    CONST jointtarget CHANGETOOL:=[[90,0,0,0,-40,0],[9E+09,9E+09,9E+09,9E+09,9E+09,9E+09]];
    TASK PERS wobjdata Pastel_2:=[FALSE,TRUE,"",[[750.001,-195.812,542.432],[0.999786,0.010364,-0.0179194,-3.3711E-5]],[[-815.382,-300.105,150],[0,0.999995,0.00323001,0]]];
    VAR robtarget Target_x_2:=[[0,0,0],[1,0,0,0],[0,0,0,0],[9E+09,9E+09,9E+09,9E+09,9E+09,9E+09]];
    CONST robtarget Aproximacion_2:=[[140.364595003,1.820278874,-22.05975894],[0.119542298,0.027125582,0.159127158,0.979618492],[-1,-1,1,0],[9E+09,9E+09,9E+09,9E+09,9E+09,9E+09]];
    CONST robtarget HOME_2:=[[685.456765267,-392.846667709,72.786791828],[0.784186035,-0.51874833,0.327913883,0.091787349],[0,0,0,0],[9E+09,9E+09,9E+09,9E+09,9E+09,9E+09]];
    CONST robtarget orientacioin_posible_2:=[[21.732086873,134.538800348,-251.768323181],[0.119514706,0.027135826,0.159101077,0.979625811],[-2,0,1,0],[9E+09,9E+09,9E+09,9E+09,9E+09,9E+09]];
    CONST robtarget Target_10_2:=[[139.514118203,143.062380794,-24.987379073],[0.119542298,0.027125582,0.159127158,0.979618492],[-1,-1,1,0],[9E+09,9E+09,9E+09,9E+09,9E+09,9E+09]];
    CONST robtarget Target_20_2:=[[138.975,143.37,0],[0.119542298,0.027125582,0.159127158,0.979618492],[-1,-1,1,0],[9E+09,9E+09,9E+09,9E+09,9E+09,9E+09]];
    CONST robtarget Target_30_2:=[[133.906,143.37,0],[0.119542298,0.027125582,0.159127158,0.979618492],[-1,-1,1,0],[9E+09,9E+09,9E+09,9E+09,9E+09,9E+09]];
    CONST robtarget Target_40_2:=[[126.245,130.656,0],[0.119542298,0.027125582,0.159127158,0.979618492],[-1,-1,1,0],[9E+09,9E+09,9E+09,9E+09,9E+09,9E+09]];
    CONST robtarget Target_50_2:=[[126.245,143.37,0],[0.119542298,0.027125582,0.159127158,0.979618492],[-1,-1,1,0],[9E+09,9E+09,9E+09,9E+09,9E+09,9E+09]];
    CONST robtarget Target_60_2:=[[121.518,143.37,0],[0.119542298,0.027125582,0.159127158,0.979618492],[-1,-1,1,0],[9E+09,9E+09,9E+09,9E+09,9E+09,9E+09]];
    CONST robtarget Target_70_2:=[[121.518,124.69,0],[0.119542298,0.027125582,0.159127158,0.979618492],[-1,-1,1,0],[9E+09,9E+09,9E+09,9E+09,9E+09,9E+09]];
    CONST robtarget Target_80_2:=[[126.603,124.69,0],[0.119542298,0.027125582,0.159127158,0.979618492],[-1,-1,1,0],[9E+09,9E+09,9E+09,9E+09,9E+09,9E+09]];
    CONST robtarget Target_90_2:=[[134.248,137.371,0],[0.119542298,0.027125582,0.159127158,0.979618492],[-1,-1,1,0],[9E+09,9E+09,9E+09,9E+09,9E+09,9E+09]];
    CONST robtarget Target_100_2:=[[134.248,124.69,0],[0.119542298,0.027125582,0.159127158,0.979618492],[-1,-1,1,0],[9E+09,9E+09,9E+09,9E+09,9E+09,9E+09]];
    CONST robtarget Target_110_2:=[[138.975,124.69,0],[0.119542298,0.027125582,0.159127158,0.979618492],[-1,-1,1,0],[9E+09,9E+09,9E+09,9E+09,9E+09,9E+09]];
    CONST robtarget Target_120_2:=[[138.975,143.37,0],[0.119542298,0.027125582,0.159127158,0.979618492],[-1,-1,1,0],[9E+09,9E+09,9E+09,9E+09,9E+09,9E+09]];
    CONST robtarget Target_130_2:=[[138.975,143.37,-10],[0.119542298,0.027125582,0.159127158,0.979618492],[-1,-1,1,0],[9E+09,9E+09,9E+09,9E+09,9E+09,9E+09]];
    CONST robtarget Target_140_2:=[[116.236,143.37,-10],[0.119542298,0.027125582,0.159127158,0.979618492],[-1,-1,1,0],[9E+09,9E+09,9E+09,9E+09,9E+09,9E+09]];
    CONST robtarget Target_150_2:=[[116.236,143.37,0],[0.119542298,0.027125582,0.159127158,0.979618492],[-1,-1,1,0],[9E+09,9E+09,9E+09,9E+09,9E+09,9E+09]];
    CONST robtarget Target_160_2:=[[111.069,143.37,0],[0.119542298,0.027125582,0.159127158,0.979618492],[-1,-1,1,0],[9E+09,9E+09,9E+09,9E+09,9E+09,9E+09]];
    CONST robtarget Target_170_2:=[[111.069,124.69,0],[0.119542298,0.027125582,0.159127158,0.979618492],[-1,-1,1,0],[9E+09,9E+09,9E+09,9E+09,9E+09,9E+09]];
    CONST robtarget Target_180_2:=[[116.236,124.69,0],[0.119542298,0.027125582,0.159127158,0.979618492],[-1,-1,1,0],[9E+09,9E+09,9E+09,9E+09,9E+09,9E+09]];
    CONST robtarget Target_190_2:=[[116.236,143.37,0],[0.119542298,0.027125582,0.159127158,0.979618492],[-1,-1,1,0],[9E+09,9E+09,9E+09,9E+09,9E+09,9E+09]];
    CONST robtarget Target_200_2:=[[116.236,143.37,-10],[0.119542298,0.027125582,0.159127158,0.979618492],[-1,-1,1,0],[9E+09,9E+09,9E+09,9E+09,9E+09,9E+09]];
    CONST robtarget Target_210_2:=[[88.445,137.143,-10],[0.119542298,0.027125582,0.159127158,0.979618492],[-1,-1,1,0],[9E+09,9E+09,9E+09,9E+09,9E+09,9E+09]];
    CONST robtarget Target_220_2:=[[88.445,137.143,0],[0.119542298,0.027125582,0.159127158,0.979618492],[-1,-1,1,0],[9E+09,9E+09,9E+09,9E+09,9E+09,9E+09]];
    CONST robtarget Target_230_2:=[[90.98,142.156,0],[0.119542298,0.027125582,0.159127158,0.979618492],[-1,-1,1,0],[9E+09,9E+09,9E+09,9E+09,9E+09,9E+09]];
    CONST robtarget Target_240_2:=[[96.97,143.973,0],[0.119542298,0.027125582,0.159127158,0.979618492],[-1,-1,1,0],[9E+09,9E+09,9E+09,9E+09,9E+09,9E+09]];
    CONST robtarget Target_250_2:=[[104.06,141.341,0],[0.119542298,0.027125582,0.159127158,0.979618492],[-1,-1,1,0],[9E+09,9E+09,9E+09,9E+09,9E+09,9E+09]];
    CONST robtarget Target_260_2:=[[106.62,134.046,0],[0.119542298,0.027125582,0.159127158,0.979618492],[-1,-1,1,0],[9E+09,9E+09,9E+09,9E+09,9E+09,9E+09]];
    CONST robtarget Target_270_2:=[[104.077,126.752,0],[0.119542298,0.027125582,0.159127158,0.979618492],[-1,-1,1,0],[9E+09,9E+09,9E+09,9E+09,9E+09,9E+09]];
    CONST robtarget Target_280_2:=[[96.954,124.136,0],[0.119542298,0.027125582,0.159127158,0.979618492],[-1,-1,1,0],[9E+09,9E+09,9E+09,9E+09,9E+09,9E+09]];
    CONST robtarget Target_290_2:=[[90.866,125.978,0],[0.119542298,0.027125582,0.159127158,0.979618492],[-1,-1,1,0],[9E+09,9E+09,9E+09,9E+09,9E+09,9E+09]];
    CONST robtarget Target_300_2:=[[88.201,131.178,0],[0.119542298,0.027125582,0.159127158,0.979618492],[-1,-1,1,0],[9E+09,9E+09,9E+09,9E+09,9E+09,9E+09]];
    CONST robtarget Target_310_2:=[[90.556,131.178,0],[0.119542298,0.027125582,0.159127158,0.979618492],[-1,-1,1,0],[9E+09,9E+09,9E+09,9E+09,9E+09,9E+09]];
    CONST robtarget Target_320_2:=[[92.911,131.178,0],[0.119542298,0.027125582,0.159127158,0.979618492],[-1,-1,1,0],[9E+09,9E+09,9E+09,9E+09,9E+09,9E+09]];
    CONST robtarget Target_330_2:=[[94.207,128.781,0],[0.119542298,0.027125582,0.159127158,0.979618492],[-1,-1,1,0],[9E+09,9E+09,9E+09,9E+09,9E+09,9E+09]];
    CONST robtarget Target_340_2:=[[96.937,127.885,0],[0.119542298,0.027125582,0.159127158,0.979618492],[-1,-1,1,0],[9E+09,9E+09,9E+09,9E+09,9E+09,9E+09]];
    CONST robtarget Target_350_2:=[[100.385,129.458,0],[0.119542298,0.027125582,0.159127158,0.979618492],[-1,-1,1,0],[9E+09,9E+09,9E+09,9E+09,9E+09,9E+09]];
    CONST robtarget Target_360_2:=[[101.583,134.03,0],[0.119542298,0.027125582,0.159127158,0.979618492],[-1,-1,1,0],[9E+09,9E+09,9E+09,9E+09,9E+09,9E+09]];
    CONST robtarget Target_370_2:=[[100.426,138.635,0],[0.119542298,0.027125582,0.159127158,0.979618492],[-1,-1,1,0],[9E+09,9E+09,9E+09,9E+09,9E+09,9E+09]];
    CONST robtarget Target_380_2:=[[96.937,140.175,0],[0.119542298,0.027125582,0.159127158,0.979618492],[-1,-1,1,0],[9E+09,9E+09,9E+09,9E+09,9E+09,9E+09]];
    CONST robtarget Target_390_2:=[[94.329,139.376,0],[0.119542298,0.027125582,0.159127158,0.979618492],[-1,-1,1,0],[9E+09,9E+09,9E+09,9E+09,9E+09,9E+09]];
    CONST robtarget Target_400_2:=[[93.058,137.143,0],[0.119542298,0.027125582,0.159127158,0.979618492],[-1,-1,1,0],[9E+09,9E+09,9E+09,9E+09,9E+09,9E+09]];
    CONST robtarget Target_410_2:=[[90.752,137.143,0],[0.119542298,0.027125582,0.159127158,0.979618492],[-1,-1,1,0],[9E+09,9E+09,9E+09,9E+09,9E+09,9E+09]];
    CONST robtarget Target_420_2:=[[88.445,137.143,0],[0.119542298,0.027125582,0.159127158,0.979618492],[-1,-1,1,0],[9E+09,9E+09,9E+09,9E+09,9E+09,9E+09]];
    CONST robtarget Target_430_2:=[[88.445,137.143,-10],[0.119542298,0.027125582,0.159127158,0.979618492],[-1,-1,1,0],[9E+09,9E+09,9E+09,9E+09,9E+09,9E+09]];
    CONST robtarget Target_440_2:=[[65.511,134.046,-10],[0.119542298,0.027125582,0.159127158,0.979618492],[-1,-1,1,0],[9E+09,9E+09,9E+09,9E+09,9E+09,9E+09]];
    CONST robtarget Target_450_2:=[[65.511,134.046,0],[0.119542298,0.027125582,0.159127158,0.979618492],[-1,-1,1,0],[9E+09,9E+09,9E+09,9E+09,9E+09,9E+09]];
    CONST robtarget Target_460_2:=[[68.127,141.3,0],[0.119542298,0.027125582,0.159127158,0.979618492],[-1,-1,1,0],[9E+09,9E+09,9E+09,9E+09,9E+09,9E+09]];
    CONST robtarget Target_470_2:=[[75.21,143.973,0],[0.119542298,0.027125582,0.159127158,0.979618492],[-1,-1,1,0],[9E+09,9E+09,9E+09,9E+09,9E+09,9E+09]];
    CONST robtarget Target_480_2:=[[82.3,141.3,0],[0.119542298,0.027125582,0.159127158,0.979618492],[-1,-1,1,0],[9E+09,9E+09,9E+09,9E+09,9E+09,9E+09]];
    CONST robtarget Target_490_2:=[[84.908,134.046,0],[0.119542298,0.027125582,0.159127158,0.979618492],[-1,-1,1,0],[9E+09,9E+09,9E+09,9E+09,9E+09,9E+09]];
    CONST robtarget Target_500_2:=[[82.3,126.809,0],[0.119542298,0.027125582,0.159127158,0.979618492],[-1,-1,1,0],[9E+09,9E+09,9E+09,9E+09,9E+09,9E+09]];
    CONST robtarget Target_510_2:=[[75.21,124.136,0],[0.119542298,0.027125582,0.159127158,0.979618492],[-1,-1,1,0],[9E+09,9E+09,9E+09,9E+09,9E+09,9E+09]];
    CONST robtarget Target_520_2:=[[68.119,126.809,0],[0.119542298,0.027125582,0.159127158,0.979618492],[-1,-1,1,0],[9E+09,9E+09,9E+09,9E+09,9E+09,9E+09]];
    CONST robtarget Target_530_2:=[[65.511,134.046,0],[0.119542298,0.027125582,0.159127158,0.979618492],[-1,-1,1,0],[9E+09,9E+09,9E+09,9E+09,9E+09,9E+09]];
    CONST robtarget Target_540_2:=[[65.511,134.046,-10],[0.119542298,0.027125582,0.159127158,0.979618492],[-1,-1,1,0],[9E+09,9E+09,9E+09,9E+09,9E+09,9E+09]];
    CONST robtarget Target_550_2:=[[71.298,134.046,-10],[0.119542298,0.027125582,0.159127158,0.979618492],[-1,-1,1,0],[9E+09,9E+09,9E+09,9E+09,9E+09,9E+09]];
    CONST robtarget Target_560_2:=[[71.298,134.046,0],[0.119542298,0.027125582,0.159127158,0.979618492],[-1,-1,1,0],[9E+09,9E+09,9E+09,9E+09,9E+09,9E+09]];
    CONST robtarget Target_570_2:=[[72.235,129.865,0],[0.119542298,0.027125582,0.159127158,0.979618492],[-1,-1,1,0],[9E+09,9E+09,9E+09,9E+09,9E+09,9E+09]];
    CONST robtarget Target_580_2:=[[75.193,128.537,0],[0.119542298,0.027125582,0.159127158,0.979618492],[-1,-1,1,0],[9E+09,9E+09,9E+09,9E+09,9E+09,9E+09]];
    CONST robtarget Target_590_2:=[[78.176,129.865,0],[0.119542298,0.027125582,0.159127158,0.979618492],[-1,-1,1,0],[9E+09,9E+09,9E+09,9E+09,9E+09,9E+09]];
    CONST robtarget Target_600_2:=[[79.122,134.046,0],[0.119542298,0.027125582,0.159127158,0.979618492],[-1,-1,1,0],[9E+09,9E+09,9E+09,9E+09,9E+09,9E+09]];
    CONST robtarget Target_610_2:=[[78.176,138.227,0],[0.119542298,0.027125582,0.159127158,0.979618492],[-1,-1,1,0],[9E+09,9E+09,9E+09,9E+09,9E+09,9E+09]];
    CONST robtarget Target_620_2:=[[75.193,139.556,0],[0.119542298,0.027125582,0.159127158,0.979618492],[-1,-1,1,0],[9E+09,9E+09,9E+09,9E+09,9E+09,9E+09]];
    CONST robtarget Target_630_2:=[[72.235,138.227,0],[0.119542298,0.027125582,0.159127158,0.979618492],[-1,-1,1,0],[9E+09,9E+09,9E+09,9E+09,9E+09,9E+09]];
    CONST robtarget Target_640_2:=[[71.298,134.046,0],[0.119542298,0.027125582,0.159127158,0.979618492],[-1,-1,1,0],[9E+09,9E+09,9E+09,9E+09,9E+09,9E+09]];
    CONST robtarget Target_650_2:=[[71.298,134.046,-10],[0.119542298,0.027125582,0.159127158,0.979618492],[-1,-1,1,0],[9E+09,9E+09,9E+09,9E+09,9E+09,9E+09]];
    CONST robtarget Target_660_2:=[[61.192,143.37,-10],[0.119542298,0.027125582,0.159127158,0.979618492],[-1,-1,1,0],[9E+09,9E+09,9E+09,9E+09,9E+09,9E+09]];
    CONST robtarget Target_670_2:=[[61.192,143.37,0],[0.119542298,0.027125582,0.159127158,0.979618492],[-1,-1,1,0],[9E+09,9E+09,9E+09,9E+09,9E+09,9E+09]];
    CONST robtarget Target_680_2:=[[56.139,143.37,0],[0.119542298,0.027125582,0.159127158,0.979618492],[-1,-1,1,0],[9E+09,9E+09,9E+09,9E+09,9E+09,9E+09]];
    CONST robtarget Target_690_2:=[[56.139,128.7,0],[0.119542298,0.027125582,0.159127158,0.979618492],[-1,-1,1,0],[9E+09,9E+09,9E+09,9E+09,9E+09,9E+09]];
    CONST robtarget Target_700_2:=[[47.402,128.7,0],[0.119542298,0.027125582,0.159127158,0.979618492],[-1,-1,1,0],[9E+09,9E+09,9E+09,9E+09,9E+09,9E+09]];
    CONST robtarget Target_710_2:=[[47.402,124.69,0],[0.119542298,0.027125582,0.159127158,0.979618492],[-1,-1,1,0],[9E+09,9E+09,9E+09,9E+09,9E+09,9E+09]];
    CONST robtarget Target_720_2:=[[61.192,124.69,0],[0.119542298,0.027125582,0.159127158,0.979618492],[-1,-1,1,0],[9E+09,9E+09,9E+09,9E+09,9E+09,9E+09]];
    CONST robtarget Target_730_2:=[[61.192,143.37,0],[0.119542298,0.027125582,0.159127158,0.979618492],[-1,-1,1,0],[9E+09,9E+09,9E+09,9E+09,9E+09,9E+09]];
    CONST robtarget Target_740_2:=[[61.192,143.37,-10],[0.119542298,0.027125582,0.159127158,0.979618492],[-1,-1,1,0],[9E+09,9E+09,9E+09,9E+09,9E+09,9E+09]];
    CONST robtarget Target_750_2:=[[38.567,143.37,-10],[0.119542298,0.027125582,0.159127158,0.979618492],[-1,-1,1,0],[9E+09,9E+09,9E+09,9E+09,9E+09,9E+09]];
    CONST robtarget Target_760_2:=[[38.567,143.37,0],[0.119542298,0.027125582,0.159127158,0.979618492],[-1,-1,1,0],[9E+09,9E+09,9E+09,9E+09,9E+09,9E+09]];
    CONST robtarget Target_770_2:=[[33.025,143.37,0],[0.119542298,0.027125582,0.159127158,0.979618492],[-1,-1,1,0],[9E+09,9E+09,9E+09,9E+09,9E+09,9E+09]];
    CONST robtarget Target_780_2:=[[26.424,124.69,0],[0.119542298,0.027125582,0.159127158,0.979618492],[-1,-1,1,0],[9E+09,9E+09,9E+09,9E+09,9E+09,9E+09]];
    CONST robtarget Target_790_2:=[[31.412,124.69,0],[0.119542298,0.027125582,0.159127158,0.979618492],[-1,-1,1,0],[9E+09,9E+09,9E+09,9E+09,9E+09,9E+09]];
    CONST robtarget Target_800_2:=[[32.178,127.331,0],[0.119542298,0.027125582,0.159127158,0.979618492],[-1,-1,1,0],[9E+09,9E+09,9E+09,9E+09,9E+09,9E+09]];
    CONST robtarget Target_810_2:=[[39.464,127.331,0],[0.119542298,0.027125582,0.159127158,0.979618492],[-1,-1,1,0],[9E+09,9E+09,9E+09,9E+09,9E+09,9E+09]];
    CONST robtarget Target_820_2:=[[40.181,124.69,0],[0.119542298,0.027125582,0.159127158,0.979618492],[-1,-1,1,0],[9E+09,9E+09,9E+09,9E+09,9E+09,9E+09]];
    CONST robtarget Target_830_2:=[[45.169,124.69,0],[0.119542298,0.027125582,0.159127158,0.979618492],[-1,-1,1,0],[9E+09,9E+09,9E+09,9E+09,9E+09,9E+09]];
    CONST robtarget Target_840_2:=[[38.567,143.37,0],[0.119542298,0.027125582,0.159127158,0.979618492],[-1,-1,1,0],[9E+09,9E+09,9E+09,9E+09,9E+09,9E+09]];
    CONST robtarget Target_850_2:=[[38.567,143.37,-10],[0.119542298,0.027125582,0.159127158,0.979618492],[-1,-1,1,0],[9E+09,9E+09,9E+09,9E+09,9E+09,9E+09]];
    CONST robtarget Target_860_2:=[[35.796,138.464,-10],[0.119542298,0.027125582,0.159127158,0.979618492],[-1,-1,1,0],[9E+09,9E+09,9E+09,9E+09,9E+09,9E+09]];
    CONST robtarget Target_870_2:=[[35.796,138.464,0],[0.119542298,0.027125582,0.159127158,0.979618492],[-1,-1,1,0],[9E+09,9E+09,9E+09,9E+09,9E+09,9E+09]];
    CONST robtarget Target_880_2:=[[37.834,130.884,0],[0.119542298,0.027125582,0.159127158,0.979618492],[-1,-1,1,0],[9E+09,9E+09,9E+09,9E+09,9E+09,9E+09]];
    CONST robtarget Target_890_2:=[[33.791,130.884,0],[0.119542298,0.027125582,0.159127158,0.979618492],[-1,-1,1,0],[9E+09,9E+09,9E+09,9E+09,9E+09,9E+09]];
    CONST robtarget Target_900_2:=[[35.796,138.464,0],[0.119542298,0.027125582,0.159127158,0.979618492],[-1,-1,1,0],[9E+09,9E+09,9E+09,9E+09,9E+09,9E+09]];
    CONST robtarget Target_910_2:=[[35.796,138.464,-10],[0.119542298,0.027125582,0.159127158,0.979618492],[-1,-1,1,0],[9E+09,9E+09,9E+09,9E+09,9E+09,9E+09]];
    CONST robtarget Target_920_2:=[[8.038,138.936,-10],[0.119542298,0.027125582,0.159127158,0.979618492],[-1,-1,1,0],[9E+09,9E+09,9E+09,9E+09,9E+09,9E+09]];
    CONST robtarget Target_930_2:=[[8.038,138.936,0],[0.119542298,0.027125582,0.159127158,0.979618492],[-1,-1,1,0],[9E+09,9E+09,9E+09,9E+09,9E+09,9E+09]];
    CONST robtarget Target_940_2:=[[10.58,142.702,0],[0.119542298,0.027125582,0.159127158,0.979618492],[-1,-1,1,0],[9E+09,9E+09,9E+09,9E+09,9E+09,9E+09]];
    CONST robtarget Target_950_2:=[[16.057,143.973,0],[0.119542298,0.027125582,0.159127158,0.979618492],[-1,-1,1,0],[9E+09,9E+09,9E+09,9E+09,9E+09,9E+09]];
    CONST robtarget Target_960_2:=[[21.558,142.416,0],[0.119542298,0.027125582,0.159127158,0.979618492],[-1,-1,1,0],[9E+09,9E+09,9E+09,9E+09,9E+09,9E+09]];
    CONST robtarget Target_970_2:=[[23.588,138.219,0],[0.119542298,0.027125582,0.159127158,0.979618492],[-1,-1,1,0],[9E+09,9E+09,9E+09,9E+09,9E+09,9E+09]];
    CONST robtarget Target_980_2:=[[22.267,134.812,0],[0.119542298,0.027125582,0.159127158,0.979618492],[-1,-1,1,0],[9E+09,9E+09,9E+09,9E+09,9E+09,9E+09]];
    CONST robtarget Target_990_2:=[[16.611,132.4,0],[0.119542298,0.027125582,0.159127158,0.979618492],[-1,-1,1,0],[9E+09,9E+09,9E+09,9E+09,9E+09,9E+09]];
    CONST robtarget Target_1000_2:=[[13.16,131.12,0],[0.119542298,0.027125582,0.159127158,0.979618492],[-1,-1,1,0],[9E+09,9E+09,9E+09,9E+09,9E+09,9E+09]];
    CONST robtarget Target_1010_2:=[[12.324,129.743,0],[0.119542298,0.027125582,0.159127158,0.979618492],[-1,-1,1,0],[9E+09,9E+09,9E+09,9E+09,9E+09,9E+09]];
    CONST robtarget Target_1020_2:=[[13.172,128.17,0],[0.119542298,0.027125582,0.159127158,0.979618492],[-1,-1,1,0],[9E+09,9E+09,9E+09,9E+09,9E+09,9E+09]];
    CONST robtarget Target_1030_2:=[[15.633,127.624,0],[0.119542298,0.027125582,0.159127158,0.979618492],[-1,-1,1,0],[9E+09,9E+09,9E+09,9E+09,9E+09,9E+09]];
    CONST robtarget Target_1040_2:=[[17.858,128.129,0],[0.119542298,0.027125582,0.159127158,0.979618492],[-1,-1,1,0],[9E+09,9E+09,9E+09,9E+09,9E+09,9E+09]];
    CONST robtarget Target_1050_2:=[[18.926,129.629,0],[0.119542298,0.027125582,0.159127158,0.979618492],[-1,-1,1,0],[9E+09,9E+09,9E+09,9E+09,9E+09,9E+09]];
    CONST robtarget Target_1060_2:=[[23.783,129.629,0],[0.119542298,0.027125582,0.159127158,0.979618492],[-1,-1,1,0],[9E+09,9E+09,9E+09,9E+09,9E+09,9E+09]];
    CONST robtarget Target_1070_2:=[[21.192,125.587,0],[0.119542298,0.027125582,0.159127158,0.979618492],[-1,-1,1,0],[9E+09,9E+09,9E+09,9E+09,9E+09,9E+09]];
    CONST robtarget Target_1080_2:=[[15.715,124.169,0],[0.119542298,0.027125582,0.159127158,0.979618492],[-1,-1,1,0],[9E+09,9E+09,9E+09,9E+09,9E+09,9E+09]];
    CONST robtarget Target_1090_2:=[[9.554,125.741,0],[0.119542298,0.027125582,0.159127158,0.979618492],[-1,-1,1,0],[9E+09,9E+09,9E+09,9E+09,9E+09,9E+09]];
    CONST robtarget Target_1100_2:=[[7.451,130.379,0],[0.119542298,0.027125582,0.159127158,0.979618492],[-1,-1,1,0],[9E+09,9E+09,9E+09,9E+09,9E+09,9E+09]];
    CONST robtarget Target_1110_2:=[[8.885,133.875,0],[0.119542298,0.027125582,0.159127158,0.979618492],[-1,-1,1,0],[9E+09,9E+09,9E+09,9E+09,9E+09,9E+09]];
    CONST robtarget Target_1120_2:=[[15.03,136.328,0],[0.119542298,0.027125582,0.159127158,0.979618492],[-1,-1,1,0],[9E+09,9E+09,9E+09,9E+09,9E+09,9E+09]];
    CONST robtarget Target_1130_2:=[[17.85,137.412,0],[0.119542298,0.027125582,0.159127158,0.979618492],[-1,-1,1,0],[9E+09,9E+09,9E+09,9E+09,9E+09,9E+09]];
    CONST robtarget Target_1140_2:=[[18.698,138.773,0],[0.119542298,0.027125582,0.159127158,0.979618492],[-1,-1,1,0],[9E+09,9E+09,9E+09,9E+09,9E+09,9E+09]];
    CONST robtarget Target_1150_2:=[[17.972,140.208,0],[0.119542298,0.027125582,0.159127158,0.979618492],[-1,-1,1,0],[9E+09,9E+09,9E+09,9E+09,9E+09,9E+09]];
    CONST robtarget Target_1160_2:=[[15.976,140.729,0],[0.119542298,0.027125582,0.159127158,0.979618492],[-1,-1,1,0],[9E+09,9E+09,9E+09,9E+09,9E+09,9E+09]];
    CONST robtarget Target_1170_2:=[[13.889,140.265,0],[0.119542298,0.027125582,0.159127158,0.979618492],[-1,-1,1,0],[9E+09,9E+09,9E+09,9E+09,9E+09,9E+09]];
    CONST robtarget Target_1180_2:=[[12.879,138.936,0],[0.119542298,0.027125582,0.159127158,0.979618492],[-1,-1,1,0],[9E+09,9E+09,9E+09,9E+09,9E+09,9E+09]];
    CONST robtarget Target_1190_2:=[[8.038,138.936,0],[0.119542298,0.027125582,0.159127158,0.979618492],[-1,-1,1,0],[9E+09,9E+09,9E+09,9E+09,9E+09,9E+09]];
    CONST robtarget Target_1200_2:=[[8.038,138.936,-10],[0.119542298,0.027125582,0.159127158,0.979618492],[-1,-1,1,0],[9E+09,9E+09,9E+09,9E+09,9E+09,9E+09]];
    CONST robtarget Target_1210_2:=[[113.571,103.208,-10],[0.119542298,0.027125582,0.159127158,0.979618492],[-1,-1,1,0],[9E+09,9E+09,9E+09,9E+09,9E+09,9E+09]];
    CONST robtarget Target_1220_2:=[[113.571,103.208,0],[0.119542298,0.027125582,0.159127158,0.979618492],[-1,-1,1,0],[9E+09,9E+09,9E+09,9E+09,9E+09,9E+09]];
    CONST robtarget Target_1230_2:=[[116.106,108.22,0],[0.119542298,0.027125582,0.159127158,0.979618492],[-1,-1,1,0],[9E+09,9E+09,9E+09,9E+09,9E+09,9E+09]];
    CONST robtarget Target_1240_2:=[[122.096,110.037,0],[0.119542298,0.027125582,0.159127158,0.979618492],[-1,-1,1,0],[9E+09,9E+09,9E+09,9E+09,9E+09,9E+09]];
    CONST robtarget Target_1250_2:=[[129.187,107.405,0],[0.119542298,0.027125582,0.159127158,0.979618492],[-1,-1,1,0],[9E+09,9E+09,9E+09,9E+09,9E+09,9E+09]];
    CONST robtarget Target_1260_2:=[[131.746,100.111,0],[0.119542298,0.027125582,0.159127158,0.979618492],[-1,-1,1,0],[9E+09,9E+09,9E+09,9E+09,9E+09,9E+09]];
    CONST robtarget Target_1270_2:=[[129.203,92.817,0],[0.119542298,0.027125582,0.159127158,0.979618492],[-1,-1,1,0],[9E+09,9E+09,9E+09,9E+09,9E+09,9E+09]];
    CONST robtarget Target_1280_2:=[[122.08,90.2,0],[0.119542298,0.027125582,0.159127158,0.979618492],[-1,-1,1,0],[9E+09,9E+09,9E+09,9E+09,9E+09,9E+09]];
    CONST robtarget Target_1290_2:=[[115.992,92.042,0],[0.119542298,0.027125582,0.159127158,0.979618492],[-1,-1,1,0],[9E+09,9E+09,9E+09,9E+09,9E+09,9E+09]];
    CONST robtarget Target_1300_2:=[[113.327,97.242,0],[0.119542298,0.027125582,0.159127158,0.979618492],[-1,-1,1,0],[9E+09,9E+09,9E+09,9E+09,9E+09,9E+09]];
    CONST robtarget Target_1310_2:=[[118.038,97.242,0],[0.119542298,0.027125582,0.159127158,0.979618492],[-1,-1,1,0],[9E+09,9E+09,9E+09,9E+09,9E+09,9E+09]];
    CONST robtarget Target_1320_2:=[[119.333,94.846,0],[0.119542298,0.027125582,0.159127158,0.979618492],[-1,-1,1,0],[9E+09,9E+09,9E+09,9E+09,9E+09,9E+09]];
    CONST robtarget Target_1330_2:=[[122.064,93.949,0],[0.119542298,0.027125582,0.159127158,0.979618492],[-1,-1,1,0],[9E+09,9E+09,9E+09,9E+09,9E+09,9E+09]];
    CONST robtarget Target_1340_2:=[[125.511,95.522,0],[0.119542298,0.027125582,0.159127158,0.979618492],[-1,-1,1,0],[9E+09,9E+09,9E+09,9E+09,9E+09,9E+09]];
    CONST robtarget Target_1350_2:=[[126.709,100.094,0],[0.119542298,0.027125582,0.159127158,0.979618492],[-1,-1,1,0],[9E+09,9E+09,9E+09,9E+09,9E+09,9E+09]];
    CONST robtarget Target_1360_2:=[[125.552,104.699,0],[0.119542298,0.027125582,0.159127158,0.979618492],[-1,-1,1,0],[9E+09,9E+09,9E+09,9E+09,9E+09,9E+09]];
    CONST robtarget Target_1370_2:=[[122.064,106.239,0],[0.119542298,0.027125582,0.159127158,0.979618492],[-1,-1,1,0],[9E+09,9E+09,9E+09,9E+09,9E+09,9E+09]];
    CONST robtarget Target_1380_2:=[[119.456,105.441,0],[0.119542298,0.027125582,0.159127158,0.979618492],[-1,-1,1,0],[9E+09,9E+09,9E+09,9E+09,9E+09,9E+09]];
    CONST robtarget Target_1390_2:=[[118.184,103.208,0],[0.119542298,0.027125582,0.159127158,0.979618492],[-1,-1,1,0],[9E+09,9E+09,9E+09,9E+09,9E+09,9E+09]];
    CONST robtarget Target_1400_2:=[[113.571,103.208,0],[0.119542298,0.027125582,0.159127158,0.979618492],[-1,-1,1,0],[9E+09,9E+09,9E+09,9E+09,9E+09,9E+09]];
    CONST robtarget Target_1410_2:=[[113.571,103.208,-10],[0.119542298,0.027125582,0.159127158,0.979618492],[-1,-1,1,0],[9E+09,9E+09,9E+09,9E+09,9E+09,9E+09]];
    CONST robtarget Target_1420_2:=[[98.771,109.434,-10],[0.119542298,0.027125582,0.159127158,0.979618492],[-1,-1,1,0],[9E+09,9E+09,9E+09,9E+09,9E+09,9E+09]];
    CONST robtarget Target_1430_2:=[[98.771,109.434,0],[0.119542298,0.027125582,0.159127158,0.979618492],[-1,-1,1,0],[9E+09,9E+09,9E+09,9E+09,9E+09,9E+09]];
    CONST robtarget Target_1440_2:=[[92.17,90.755,0],[0.119542298,0.027125582,0.159127158,0.979618492],[-1,-1,1,0],[9E+09,9E+09,9E+09,9E+09,9E+09,9E+09]];
    CONST robtarget Target_1450_2:=[[97.157,90.755,0],[0.119542298,0.027125582,0.159127158,0.979618492],[-1,-1,1,0],[9E+09,9E+09,9E+09,9E+09,9E+09,9E+09]];
    CONST robtarget Target_1460_2:=[[97.924,93.395,0],[0.119542298,0.027125582,0.159127158,0.979618492],[-1,-1,1,0],[9E+09,9E+09,9E+09,9E+09,9E+09,9E+09]];
    CONST robtarget Target_1470_2:=[[105.21,93.395,0],[0.119542298,0.027125582,0.159127158,0.979618492],[-1,-1,1,0],[9E+09,9E+09,9E+09,9E+09,9E+09,9E+09]];
    CONST robtarget Target_1480_2:=[[105.927,90.755,0],[0.119542298,0.027125582,0.159127158,0.979618492],[-1,-1,1,0],[9E+09,9E+09,9E+09,9E+09,9E+09,9E+09]];
    CONST robtarget Target_1490_2:=[[110.915,90.755,0],[0.119542298,0.027125582,0.159127158,0.979618492],[-1,-1,1,0],[9E+09,9E+09,9E+09,9E+09,9E+09,9E+09]];
    CONST robtarget Target_1500_2:=[[104.313,109.434,0],[0.119542298,0.027125582,0.159127158,0.979618492],[-1,-1,1,0],[9E+09,9E+09,9E+09,9E+09,9E+09,9E+09]];
    CONST robtarget Target_1510_2:=[[98.771,109.434,0],[0.119542298,0.027125582,0.159127158,0.979618492],[-1,-1,1,0],[9E+09,9E+09,9E+09,9E+09,9E+09,9E+09]];
    CONST robtarget Target_1520_2:=[[98.771,109.434,-10],[0.119542298,0.027125582,0.159127158,0.979618492],[-1,-1,1,0],[9E+09,9E+09,9E+09,9E+09,9E+09,9E+09]];
    CONST robtarget Target_1530_2:=[[101.542,104.528,-10],[0.119542298,0.027125582,0.159127158,0.979618492],[-1,-1,1,0],[9E+09,9E+09,9E+09,9E+09,9E+09,9E+09]];
    CONST robtarget Target_1540_2:=[[101.542,104.528,0],[0.119542298,0.027125582,0.159127158,0.979618492],[-1,-1,1,0],[9E+09,9E+09,9E+09,9E+09,9E+09,9E+09]];
    CONST robtarget Target_1550_2:=[[103.58,96.949,0],[0.119542298,0.027125582,0.159127158,0.979618492],[-1,-1,1,0],[9E+09,9E+09,9E+09,9E+09,9E+09,9E+09]];
    CONST robtarget Target_1560_2:=[[99.537,96.949,0],[0.119542298,0.027125582,0.159127158,0.979618492],[-1,-1,1,0],[9E+09,9E+09,9E+09,9E+09,9E+09,9E+09]];
    CONST robtarget Target_1570_2:=[[101.542,104.528,0],[0.119542298,0.027125582,0.159127158,0.979618492],[-1,-1,1,0],[9E+09,9E+09,9E+09,9E+09,9E+09,9E+09]];
    CONST robtarget Target_1580_2:=[[101.542,104.528,-10],[0.119542298,0.027125582,0.159127158,0.979618492],[-1,-1,1,0],[9E+09,9E+09,9E+09,9E+09,9E+09,9E+09]];
    CONST robtarget Target_1590_2:=[[88.747,109.434,-10],[0.119542298,0.027125582,0.159127158,0.979618492],[-1,-1,1,0],[9E+09,9E+09,9E+09,9E+09,9E+09,9E+09]];
    CONST robtarget Target_1600_2:=[[88.747,109.434,0],[0.119542298,0.027125582,0.159127158,0.979618492],[-1,-1,1,0],[9E+09,9E+09,9E+09,9E+09,9E+09,9E+09]];
    CONST robtarget Target_1610_2:=[[88.747,90.755,0],[0.119542298,0.027125582,0.159127158,0.979618492],[-1,-1,1,0],[9E+09,9E+09,9E+09,9E+09,9E+09,9E+09]];
    CONST robtarget Target_1620_2:=[[84.297,90.755,0],[0.119542298,0.027125582,0.159127158,0.979618492],[-1,-1,1,0],[9E+09,9E+09,9E+09,9E+09,9E+09,9E+09]];
    CONST robtarget Target_1630_2:=[[84.297,105.848,0],[0.119542298,0.027125582,0.159127158,0.979618492],[-1,-1,1,0],[9E+09,9E+09,9E+09,9E+09,9E+09,9E+09]];
    CONST robtarget Target_1640_2:=[[83.743,105.848,0],[0.119542298,0.027125582,0.159127158,0.979618492],[-1,-1,1,0],[9E+09,9E+09,9E+09,9E+09,9E+09,9E+09]];
    CONST robtarget Target_1650_2:=[[79.88,90.755,0],[0.119542298,0.027125582,0.159127158,0.979618492],[-1,-1,1,0],[9E+09,9E+09,9E+09,9E+09,9E+09,9E+09]];
    CONST robtarget Target_1660_2:=[[76.424,90.755,0],[0.119542298,0.027125582,0.159127158,0.979618492],[-1,-1,1,0],[9E+09,9E+09,9E+09,9E+09,9E+09,9E+09]];
    CONST robtarget Target_1670_2:=[[72.626,105.848,0],[0.119542298,0.027125582,0.159127158,0.979618492],[-1,-1,1,0],[9E+09,9E+09,9E+09,9E+09,9E+09,9E+09]];
    CONST robtarget Target_1680_2:=[[71.941,105.848,0],[0.119542298,0.027125582,0.159127158,0.979618492],[-1,-1,1,0],[9E+09,9E+09,9E+09,9E+09,9E+09,9E+09]];
    CONST robtarget Target_1690_2:=[[71.941,90.755,0],[0.119542298,0.027125582,0.159127158,0.979618492],[-1,-1,1,0],[9E+09,9E+09,9E+09,9E+09,9E+09,9E+09]];
    CONST robtarget Target_1700_2:=[[67.557,90.755,0],[0.119542298,0.027125582,0.159127158,0.979618492],[-1,-1,1,0],[9E+09,9E+09,9E+09,9E+09,9E+09,9E+09]];
    CONST robtarget Target_1710_2:=[[67.557,109.434,0],[0.119542298,0.027125582,0.159127158,0.979618492],[-1,-1,1,0],[9E+09,9E+09,9E+09,9E+09,9E+09,9E+09]];
    CONST robtarget Target_1720_2:=[[74.175,109.434,0],[0.119542298,0.027125582,0.159127158,0.979618492],[-1,-1,1,0],[9E+09,9E+09,9E+09,9E+09,9E+09,9E+09]];
    CONST robtarget Target_1730_2:=[[78.152,95.482,0],[0.119542298,0.027125582,0.159127158,0.979618492],[-1,-1,1,0],[9E+09,9E+09,9E+09,9E+09,9E+09,9E+09]];
    CONST robtarget Target_1740_2:=[[82.113,109.434,0],[0.119542298,0.027125582,0.159127158,0.979618492],[-1,-1,1,0],[9E+09,9E+09,9E+09,9E+09,9E+09,9E+09]];
    CONST robtarget Target_1750_2:=[[88.747,109.434,0],[0.119542298,0.027125582,0.159127158,0.979618492],[-1,-1,1,0],[9E+09,9E+09,9E+09,9E+09,9E+09,9E+09]];
    CONST robtarget Target_1760_2:=[[88.747,109.434,-10],[0.119542298,0.027125582,0.159127158,0.979618492],[-1,-1,1,0],[9E+09,9E+09,9E+09,9E+09,9E+09,9E+09]];
    CONST robtarget Target_1770_2:=[[62.308,109.434,-10],[0.119542298,0.027125582,0.159127158,0.979618492],[-1,-1,1,0],[9E+09,9E+09,9E+09,9E+09,9E+09,9E+09]];
    CONST robtarget Target_1780_2:=[[62.308,109.434,0],[0.119542298,0.027125582,0.159127158,0.979618492],[-1,-1,1,0],[9E+09,9E+09,9E+09,9E+09,9E+09,9E+09]];
    CONST robtarget Target_1790_2:=[[62.308,90.755,0],[0.119542298,0.027125582,0.159127158,0.979618492],[-1,-1,1,0],[9E+09,9E+09,9E+09,9E+09,9E+09,9E+09]];
    CONST robtarget Target_1800_2:=[[57.141,90.755,0],[0.119542298,0.027125582,0.159127158,0.979618492],[-1,-1,1,0],[9E+09,9E+09,9E+09,9E+09,9E+09,9E+09]];
    CONST robtarget Target_1810_2:=[[57.141,109.434,0],[0.119542298,0.027125582,0.159127158,0.979618492],[-1,-1,1,0],[9E+09,9E+09,9E+09,9E+09,9E+09,9E+09]];
    CONST robtarget Target_1820_2:=[[62.308,109.434,0],[0.119542298,0.027125582,0.159127158,0.979618492],[-1,-1,1,0],[9E+09,9E+09,9E+09,9E+09,9E+09,9E+09]];
    CONST robtarget Target_1830_2:=[[62.308,109.434,-10],[0.119542298,0.027125582,0.159127158,0.979618492],[-1,-1,1,0],[9E+09,9E+09,9E+09,9E+09,9E+09,9E+09]];
    CONST robtarget Target_1840_2:=[[51.86,109.434,-10],[0.119542298,0.027125582,0.159127158,0.979618492],[-1,-1,1,0],[9E+09,9E+09,9E+09,9E+09,9E+09,9E+09]];
    CONST robtarget Target_1850_2:=[[51.86,109.434,0],[0.119542298,0.027125582,0.159127158,0.979618492],[-1,-1,1,0],[9E+09,9E+09,9E+09,9E+09,9E+09,9E+09]];
    CONST robtarget Target_1860_2:=[[51.86,90.755,0],[0.119542298,0.027125582,0.159127158,0.979618492],[-1,-1,1,0],[9E+09,9E+09,9E+09,9E+09,9E+09,9E+09]];
    CONST robtarget Target_1870_2:=[[38.07,90.755,0],[0.119542298,0.027125582,0.159127158,0.979618492],[-1,-1,1,0],[9E+09,9E+09,9E+09,9E+09,9E+09,9E+09]];
    CONST robtarget Target_1880_2:=[[38.07,94.764,0],[0.119542298,0.027125582,0.159127158,0.979618492],[-1,-1,1,0],[9E+09,9E+09,9E+09,9E+09,9E+09,9E+09]];
    CONST robtarget Target_1890_2:=[[46.807,94.764,0],[0.119542298,0.027125582,0.159127158,0.979618492],[-1,-1,1,0],[9E+09,9E+09,9E+09,9E+09,9E+09,9E+09]];
    CONST robtarget Target_1900_2:=[[46.807,109.434,0],[0.119542298,0.027125582,0.159127158,0.979618492],[-1,-1,1,0],[9E+09,9E+09,9E+09,9E+09,9E+09,9E+09]];
    CONST robtarget Target_1910_2:=[[51.86,109.434,0],[0.119542298,0.027125582,0.159127158,0.979618492],[-1,-1,1,0],[9E+09,9E+09,9E+09,9E+09,9E+09,9E+09]];
    CONST robtarget Target_1920_2:=[[51.86,109.434,-10],[0.119542298,0.027125582,0.159127158,0.979618492],[-1,-1,1,0],[9E+09,9E+09,9E+09,9E+09,9E+09,9E+09]];
    CONST robtarget Target_1930_2:=[[25.242,106.256,-10],[0.119542298,0.027125582,0.159127158,0.979618492],[-1,-1,1,0],[9E+09,9E+09,9E+09,9E+09,9E+09,9E+09]];
    CONST robtarget Target_1940_2:=[[25.242,106.256,0],[0.119542298,0.027125582,0.159127158,0.979618492],[-1,-1,1,0],[9E+09,9E+09,9E+09,9E+09,9E+09,9E+09]];
    CONST robtarget Target_1950_2:=[[28.739,104.772,0],[0.119542298,0.027125582,0.159127158,0.979618492],[-1,-1,1,0],[9E+09,9E+09,9E+09,9E+09,9E+09,9E+09]];
    CONST robtarget Target_1960_2:=[[29.855,100.111,0],[0.119542298,0.027125582,0.159127158,0.979618492],[-1,-1,1,0],[9E+09,9E+09,9E+09,9E+09,9E+09,9E+09]];
    CONST robtarget Target_1970_2:=[[28.739,95.449,0],[0.119542298,0.027125582,0.159127158,0.979618492],[-1,-1,1,0],[9E+09,9E+09,9E+09,9E+09,9E+09,9E+09]];
    CONST robtarget Target_1980_2:=[[25.242,93.966,0],[0.119542298,0.027125582,0.159127158,0.979618492],[-1,-1,1,0],[9E+09,9E+09,9E+09,9E+09,9E+09,9E+09]];
    CONST robtarget Target_1990_2:=[[21.754,95.441,0],[0.119542298,0.027125582,0.159127158,0.979618492],[-1,-1,1,0],[9E+09,9E+09,9E+09,9E+09,9E+09,9E+09]];
    CONST robtarget Target_2000_2:=[[20.646,100.111,0],[0.119542298,0.027125582,0.159127158,0.979618492],[-1,-1,1,0],[9E+09,9E+09,9E+09,9E+09,9E+09,9E+09]];
    CONST robtarget Target_2010_2:=[[21.754,104.772,0],[0.119542298,0.027125582,0.159127158,0.979618492],[-1,-1,1,0],[9E+09,9E+09,9E+09,9E+09,9E+09,9E+09]];
    CONST robtarget Target_2020_2:=[[25.242,106.256,0],[0.119542298,0.027125582,0.159127158,0.979618492],[-1,-1,1,0],[9E+09,9E+09,9E+09,9E+09,9E+09,9E+09]];
    CONST robtarget Target_2030_2:=[[25.242,106.256,-10],[0.119542298,0.027125582,0.159127158,0.979618492],[-1,-1,1,0],[9E+09,9E+09,9E+09,9E+09,9E+09,9E+09]];
    CONST robtarget Target_2040_2:=[[25.258,110.037,-10],[0.119542298,0.027125582,0.159127158,0.979618492],[-1,-1,1,0],[9E+09,9E+09,9E+09,9E+09,9E+09,9E+09]];
    CONST robtarget Target_2050_2:=[[25.258,110.037,0],[0.119542298,0.027125582,0.159127158,0.979618492],[-1,-1,1,0],[9E+09,9E+09,9E+09,9E+09,9E+09,9E+09]];
    CONST robtarget Target_2060_2:=[[18.176,107.364,0],[0.119542298,0.027125582,0.159127158,0.979618492],[-1,-1,1,0],[9E+09,9E+09,9E+09,9E+09,9E+09,9E+09]];
    CONST robtarget Target_2070_2:=[[15.56,100.111,0],[0.119542298,0.027125582,0.159127158,0.979618492],[-1,-1,1,0],[9E+09,9E+09,9E+09,9E+09,9E+09,9E+09]];
    CONST robtarget Target_2080_2:=[[18.168,92.874,0],[0.119542298,0.027125582,0.159127158,0.979618492],[-1,-1,1,0],[9E+09,9E+09,9E+09,9E+09,9E+09,9E+09]];
    CONST robtarget Target_2090_2:=[[25.258,90.2,0],[0.119542298,0.027125582,0.159127158,0.979618492],[-1,-1,1,0],[9E+09,9E+09,9E+09,9E+09,9E+09,9E+09]];
    CONST robtarget Target_2100_2:=[[32.349,92.874,0],[0.119542298,0.027125582,0.159127158,0.979618492],[-1,-1,1,0],[9E+09,9E+09,9E+09,9E+09,9E+09,9E+09]];
    CONST robtarget Target_2110_2:=[[34.957,100.111,0],[0.119542298,0.027125582,0.159127158,0.979618492],[-1,-1,1,0],[9E+09,9E+09,9E+09,9E+09,9E+09,9E+09]];
    CONST robtarget Target_2120_2:=[[32.349,107.364,0],[0.119542298,0.027125582,0.159127158,0.979618492],[-1,-1,1,0],[9E+09,9E+09,9E+09,9E+09,9E+09,9E+09]];
    CONST robtarget Target_2130_2:=[[25.258,110.037,0],[0.119542298,0.027125582,0.159127158,0.979618492],[-1,-1,1,0],[9E+09,9E+09,9E+09,9E+09,9E+09,9E+09]];
    CONST robtarget Target_2140_2:=[[25.258,110.037,-10],[0.119542298,0.027125582,0.159127158,0.979618492],[-1,-1,1,0],[9E+09,9E+09,9E+09,9E+09,9E+09,9E+09]];
    CONST robtarget Target_2150_2:=[[120.369,69.924,-10],[0.119542298,0.027125582,0.159127158,0.979618492],[-1,-1,1,0],[9E+09,9E+09,9E+09,9E+09,9E+09,9E+09]];
    CONST robtarget Target_2160_2:=[[120.369,69.924,0],[0.119542298,0.027125582,0.159127158,0.979618492],[-1,-1,1,0],[9E+09,9E+09,9E+09,9E+09,9E+09,9E+09]];
    CONST robtarget Target_2170_2:=[[125.21,69.924,0],[0.119542298,0.027125582,0.159127158,0.979618492],[-1,-1,1,0],[9E+09,9E+09,9E+09,9E+09,9E+09,9E+09]];
    CONST robtarget Target_2180_2:=[[126.514,71.717,0],[0.119542298,0.027125582,0.159127158,0.979618492],[-1,-1,1,0],[9E+09,9E+09,9E+09,9E+09,9E+09,9E+09]];
    CONST robtarget Target_2190_2:=[[128.763,72.337,0],[0.119542298,0.027125582,0.159127158,0.979618492],[-1,-1,1,0],[9E+09,9E+09,9E+09,9E+09,9E+09,9E+09]];
    CONST robtarget Target_2200_2:=[[132.178,70.715,0],[0.119542298,0.027125582,0.159127158,0.979618492],[-1,-1,1,0],[9E+09,9E+09,9E+09,9E+09,9E+09,9E+09]];
    CONST robtarget Target_2210_2:=[[133.376,66.061,0],[0.119542298,0.027125582,0.159127158,0.979618492],[-1,-1,1,0],[9E+09,9E+09,9E+09,9E+09,9E+09,9E+09]];
    CONST robtarget Target_2220_2:=[[132.243,61.367,0],[0.119542298,0.027125582,0.159127158,0.979618492],[-1,-1,1,0],[9E+09,9E+09,9E+09,9E+09,9E+09,9E+09]];
    CONST robtarget Target_2230_2:=[[128.763,59.834,0],[0.119542298,0.027125582,0.159127158,0.979618492],[-1,-1,1,0],[9E+09,9E+09,9E+09,9E+09,9E+09,9E+09]];
    CONST robtarget Target_2240_2:=[[125.723,60.861,0],[0.119542298,0.027125582,0.159127158,0.979618492],[-1,-1,1,0],[9E+09,9E+09,9E+09,9E+09,9E+09,9E+09]];
    CONST robtarget Target_2250_2:=[[124.46,63.486,0],[0.119542298,0.027125582,0.159127158,0.979618492],[-1,-1,1,0],[9E+09,9E+09,9E+09,9E+09,9E+09,9E+09]];
    CONST robtarget Target_2260_2:=[[125.927,63.494,0],[0.119542298,0.027125582,0.159127158,0.979618492],[-1,-1,1,0],[9E+09,9E+09,9E+09,9E+09,9E+09,9E+09]];
    CONST robtarget Target_2270_2:=[[127.394,63.502,0],[0.119542298,0.027125582,0.159127158,0.979618492],[-1,-1,1,0],[9E+09,9E+09,9E+09,9E+09,9E+09,9E+09]];
    CONST robtarget Target_2280_2:=[[127.394,66.501,0],[0.119542298,0.027125582,0.159127158,0.979618492],[-1,-1,1,0],[9E+09,9E+09,9E+09,9E+09,9E+09,9E+09]];
    CONST robtarget Target_2290_2:=[[119.961,66.501,0],[0.119542298,0.027125582,0.159127158,0.979618492],[-1,-1,1,0],[9E+09,9E+09,9E+09,9E+09,9E+09,9E+09]];
    CONST robtarget Target_2300_2:=[[119.961,56.819,0],[0.119542298,0.027125582,0.159127158,0.979618492],[-1,-1,1,0],[9E+09,9E+09,9E+09,9E+09,9E+09,9E+09]];
    CONST robtarget Target_2310_2:=[[122.928,56.819,0],[0.119542298,0.027125582,0.159127158,0.979618492],[-1,-1,1,0],[9E+09,9E+09,9E+09,9E+09,9E+09,9E+09]];
    CONST robtarget Target_2320_2:=[[123.433,59.557,0],[0.119542298,0.027125582,0.159127158,0.979618492],[-1,-1,1,0],[9E+09,9E+09,9E+09,9E+09,9E+09,9E+09]];
    CONST robtarget Target_2330_2:=[[125.78,57.129,0],[0.119542298,0.027125582,0.159127158,0.979618492],[-1,-1,1,0],[9E+09,9E+09,9E+09,9E+09,9E+09,9E+09]];
    CONST robtarget Target_2340_2:=[[129.855,56.265,0],[0.119542298,0.027125582,0.159127158,0.979618492],[-1,-1,1,0],[9E+09,9E+09,9E+09,9E+09,9E+09,9E+09]];
    CONST robtarget Target_2350_2:=[[136.155,58.938,0],[0.119542298,0.027125582,0.159127158,0.979618492],[-1,-1,1,0],[9E+09,9E+09,9E+09,9E+09,9E+09,9E+09]];
    CONST robtarget Target_2360_2:=[[138.478,66.175,0],[0.119542298,0.027125582,0.159127158,0.979618492],[-1,-1,1,0],[9E+09,9E+09,9E+09,9E+09,9E+09,9E+09]];
    CONST robtarget Target_2370_2:=[[135.91,73.469,0],[0.119542298,0.027125582,0.159127158,0.979618492],[-1,-1,1,0],[9E+09,9E+09,9E+09,9E+09,9E+09,9E+09]];
    CONST robtarget Target_2380_2:=[[128.796,76.102,0],[0.119542298,0.027125582,0.159127158,0.979618492],[-1,-1,1,0],[9E+09,9E+09,9E+09,9E+09,9E+09,9E+09]];
    CONST robtarget Target_2390_2:=[[123.148,74.48,0],[0.119542298,0.027125582,0.159127158,0.979618492],[-1,-1,1,0],[9E+09,9E+09,9E+09,9E+09,9E+09,9E+09]];
    CONST robtarget Target_2400_2:=[[120.369,69.924,0],[0.119542298,0.027125582,0.159127158,0.979618492],[-1,-1,1,0],[9E+09,9E+09,9E+09,9E+09,9E+09,9E+09]];
    CONST robtarget Target_2410_2:=[[120.369,69.924,-10],[0.119542298,0.027125582,0.159127158,0.979618492],[-1,-1,1,0],[9E+09,9E+09,9E+09,9E+09,9E+09,9E+09]];
    CONST robtarget Target_2420_2:=[[110.1,75.499,-10],[0.119542298,0.027125582,0.159127158,0.979618492],[-1,-1,1,0],[9E+09,9E+09,9E+09,9E+09,9E+09,9E+09]];
    CONST robtarget Target_2430_2:=[[110.1,75.499,0],[0.119542298,0.027125582,0.159127158,0.979618492],[-1,-1,1,0],[9E+09,9E+09,9E+09,9E+09,9E+09,9E+09]];
    CONST robtarget Target_2440_2:=[[104.558,75.499,0],[0.119542298,0.027125582,0.159127158,0.979618492],[-1,-1,1,0],[9E+09,9E+09,9E+09,9E+09,9E+09,9E+09]];
    CONST robtarget Target_2450_2:=[[97.956,56.819,0],[0.119542298,0.027125582,0.159127158,0.979618492],[-1,-1,1,0],[9E+09,9E+09,9E+09,9E+09,9E+09,9E+09]];
    CONST robtarget Target_2460_2:=[[102.944,56.819,0],[0.119542298,0.027125582,0.159127158,0.979618492],[-1,-1,1,0],[9E+09,9E+09,9E+09,9E+09,9E+09,9E+09]];
    CONST robtarget Target_2470_2:=[[103.71,59.46,0],[0.119542298,0.027125582,0.159127158,0.979618492],[-1,-1,1,0],[9E+09,9E+09,9E+09,9E+09,9E+09,9E+09]];
    CONST robtarget Target_2480_2:=[[110.996,59.46,0],[0.119542298,0.027125582,0.159127158,0.979618492],[-1,-1,1,0],[9E+09,9E+09,9E+09,9E+09,9E+09,9E+09]];
    CONST robtarget Target_2490_2:=[[111.713,56.819,0],[0.119542298,0.027125582,0.159127158,0.979618492],[-1,-1,1,0],[9E+09,9E+09,9E+09,9E+09,9E+09,9E+09]];
    CONST robtarget Target_2500_2:=[[116.701,56.819,0],[0.119542298,0.027125582,0.159127158,0.979618492],[-1,-1,1,0],[9E+09,9E+09,9E+09,9E+09,9E+09,9E+09]];
    CONST robtarget Target_2510_2:=[[110.1,75.499,0],[0.119542298,0.027125582,0.159127158,0.979618492],[-1,-1,1,0],[9E+09,9E+09,9E+09,9E+09,9E+09,9E+09]];
    CONST robtarget Target_2520_2:=[[110.1,75.499,-10],[0.119542298,0.027125582,0.159127158,0.979618492],[-1,-1,1,0],[9E+09,9E+09,9E+09,9E+09,9E+09,9E+09]];
    CONST robtarget Target_2530_2:=[[107.329,70.592,-10],[0.119542298,0.027125582,0.159127158,0.979618492],[-1,-1,1,0],[9E+09,9E+09,9E+09,9E+09,9E+09,9E+09]];
    CONST robtarget Target_2540_2:=[[107.329,70.592,0],[0.119542298,0.027125582,0.159127158,0.979618492],[-1,-1,1,0],[9E+09,9E+09,9E+09,9E+09,9E+09,9E+09]];
    CONST robtarget Target_2550_2:=[[109.366,63.013,0],[0.119542298,0.027125582,0.159127158,0.979618492],[-1,-1,1,0],[9E+09,9E+09,9E+09,9E+09,9E+09,9E+09]];
    CONST robtarget Target_2560_2:=[[105.324,63.013,0],[0.119542298,0.027125582,0.159127158,0.979618492],[-1,-1,1,0],[9E+09,9E+09,9E+09,9E+09,9E+09,9E+09]];
    CONST robtarget Target_2570_2:=[[107.329,70.592,0],[0.119542298,0.027125582,0.159127158,0.979618492],[-1,-1,1,0],[9E+09,9E+09,9E+09,9E+09,9E+09,9E+09]];
    CONST robtarget Target_2580_2:=[[107.329,70.592,-10],[0.119542298,0.027125582,0.159127158,0.979618492],[-1,-1,1,0],[9E+09,9E+09,9E+09,9E+09,9E+09,9E+09]];
    CONST robtarget Target_2590_2:=[[94.533,75.499,-10],[0.119542298,0.027125582,0.159127158,0.979618492],[-1,-1,1,0],[9E+09,9E+09,9E+09,9E+09,9E+09,9E+09]];
    CONST robtarget Target_2600_2:=[[94.533,75.499,0],[0.119542298,0.027125582,0.159127158,0.979618492],[-1,-1,1,0],[9E+09,9E+09,9E+09,9E+09,9E+09,9E+09]];
    CONST robtarget Target_2610_2:=[[86.921,75.499,0],[0.119542298,0.027125582,0.159127158,0.979618492],[-1,-1,1,0],[9E+09,9E+09,9E+09,9E+09,9E+09,9E+09]];
    CONST robtarget Target_2620_2:=[[81.379,74.944,0],[0.119542298,0.027125582,0.159127158,0.979618492],[-1,-1,1,0],[9E+09,9E+09,9E+09,9E+09,9E+09,9E+09]];
    CONST robtarget Target_2630_2:=[[79.366,73.355,0],[0.119542298,0.027125582,0.159127158,0.979618492],[-1,-1,1,0],[9E+09,9E+09,9E+09,9E+09,9E+09,9E+09]];
    CONST robtarget Target_2640_2:=[[78.624,70.804,0],[0.119542298,0.027125582,0.159127158,0.979618492],[-1,-1,1,0],[9E+09,9E+09,9E+09,9E+09,9E+09,9E+09]];
    CONST robtarget Target_2650_2:=[[79.382,68.433,0],[0.119542298,0.027125582,0.159127158,0.979618492],[-1,-1,1,0],[9E+09,9E+09,9E+09,9E+09,9E+09,9E+09]];
    CONST robtarget Target_2660_2:=[[81.509,66.795,0],[0.119542298,0.027125582,0.159127158,0.979618492],[-1,-1,1,0],[9E+09,9E+09,9E+09,9E+09,9E+09,9E+09]];
    CONST robtarget Target_2670_2:=[[78.869,64.993,0],[0.119542298,0.027125582,0.159127158,0.979618492],[-1,-1,1,0],[9E+09,9E+09,9E+09,9E+09,9E+09,9E+09]];
    CONST robtarget Target_2680_2:=[[78.005,61.986,0],[0.119542298,0.027125582,0.159127158,0.979618492],[-1,-1,1,0],[9E+09,9E+09,9E+09,9E+09,9E+09,9E+09]];
    CONST robtarget Target_2690_2:=[[78.673,59.394,0],[0.119542298,0.027125582,0.159127158,0.979618492],[-1,-1,1,0],[9E+09,9E+09,9E+09,9E+09,9E+09,9E+09]];
    CONST robtarget Target_2700_2:=[[80.564,57.667,0],[0.119542298,0.027125582,0.159127158,0.979618492],[-1,-1,1,0],[9E+09,9E+09,9E+09,9E+09,9E+09,9E+09]];
    CONST robtarget Target_2710_2:=[[82.577,57.015,0],[0.119542298,0.027125582,0.159127158,0.979618492],[-1,-1,1,0],[9E+09,9E+09,9E+09,9E+09,9E+09,9E+09]];
    CONST robtarget Target_2720_2:=[[86.122,56.819,0],[0.119542298,0.027125582,0.159127158,0.979618492],[-1,-1,1,0],[9E+09,9E+09,9E+09,9E+09,9E+09,9E+09]];
    CONST robtarget Target_2730_2:=[[94.533,56.819,0],[0.119542298,0.027125582,0.159127158,0.979618492],[-1,-1,1,0],[9E+09,9E+09,9E+09,9E+09,9E+09,9E+09]];
    CONST robtarget Target_2740_2:=[[94.533,75.499,0],[0.119542298,0.027125582,0.159127158,0.979618492],[-1,-1,1,0],[9E+09,9E+09,9E+09,9E+09,9E+09,9E+09]];
    CONST robtarget Target_2750_2:=[[94.533,75.499,-10],[0.119542298,0.027125582,0.159127158,0.979618492],[-1,-1,1,0],[9E+09,9E+09,9E+09,9E+09,9E+09,9E+09]];
    CONST robtarget Target_2760_2:=[[88.991,71.652,-10],[0.119542298,0.027125582,0.159127158,0.979618492],[-1,-1,1,0],[9E+09,9E+09,9E+09,9E+09,9E+09,9E+09]];
    CONST robtarget Target_2770_2:=[[88.991,71.652,0],[0.119542298,0.027125582,0.159127158,0.979618492],[-1,-1,1,0],[9E+09,9E+09,9E+09,9E+09,9E+09,9E+09]];
    CONST robtarget Target_2780_2:=[[87.214,71.652,0],[0.119542298,0.027125582,0.159127158,0.979618492],[-1,-1,1,0],[9E+09,9E+09,9E+09,9E+09,9E+09,9E+09]];
    CONST robtarget Target_2790_2:=[[84.501,71.285,0],[0.119542298,0.027125582,0.159127158,0.979618492],[-1,-1,1,0],[9E+09,9E+09,9E+09,9E+09,9E+09,9E+09]];
    CONST robtarget Target_2800_2:=[[83.922,69.924,0],[0.119542298,0.027125582,0.159127158,0.979618492],[-1,-1,1,0],[9E+09,9E+09,9E+09,9E+09,9E+09,9E+09]];
    CONST robtarget Target_2810_2:=[[84.468,68.596,0],[0.119542298,0.027125582,0.159127158,0.979618492],[-1,-1,1,0],[9E+09,9E+09,9E+09,9E+09,9E+09,9E+09]];
    CONST robtarget Target_2820_2:=[[86.334,68.196,0],[0.119542298,0.027125582,0.159127158,0.979618492],[-1,-1,1,0],[9E+09,9E+09,9E+09,9E+09,9E+09,9E+09]];
    CONST robtarget Target_2830_2:=[[87.663,68.196,0],[0.119542298,0.027125582,0.159127158,0.979618492],[-1,-1,1,0],[9E+09,9E+09,9E+09,9E+09,9E+09,9E+09]];
    CONST robtarget Target_2840_2:=[[88.991,68.196,0],[0.119542298,0.027125582,0.159127158,0.979618492],[-1,-1,1,0],[9E+09,9E+09,9E+09,9E+09,9E+09,9E+09]];
    CONST robtarget Target_2850_2:=[[88.991,71.652,0],[0.119542298,0.027125582,0.159127158,0.979618492],[-1,-1,1,0],[9E+09,9E+09,9E+09,9E+09,9E+09,9E+09]];
    CONST robtarget Target_2860_2:=[[88.991,71.652,-10],[0.119542298,0.027125582,0.159127158,0.979618492],[-1,-1,1,0],[9E+09,9E+09,9E+09,9E+09,9E+09,9E+09]];
    CONST robtarget Target_2870_2:=[[88.991,64.545,-10],[0.119542298,0.027125582,0.159127158,0.979618492],[-1,-1,1,0],[9E+09,9E+09,9E+09,9E+09,9E+09,9E+09]];
    CONST robtarget Target_2880_2:=[[88.991,64.545,0],[0.119542298,0.027125582,0.159127158,0.979618492],[-1,-1,1,0],[9E+09,9E+09,9E+09,9E+09,9E+09,9E+09]];
    CONST robtarget Target_2890_2:=[[87.532,64.545,0],[0.119542298,0.027125582,0.159127158,0.979618492],[-1,-1,1,0],[9E+09,9E+09,9E+09,9E+09,9E+09,9E+09]];
    CONST robtarget Target_2900_2:=[[86.073,64.545,0],[0.119542298,0.027125582,0.159127158,0.979618492],[-1,-1,1,0],[9E+09,9E+09,9E+09,9E+09,9E+09,9E+09]];
    CONST robtarget Target_2910_2:=[[83.922,64.121,0],[0.119542298,0.027125582,0.159127158,0.979618492],[-1,-1,1,0],[9E+09,9E+09,9E+09,9E+09,9E+09,9E+09]];
    CONST robtarget Target_2920_2:=[[83.286,62.72,0],[0.119542298,0.027125582,0.159127158,0.979618492],[-1,-1,1,0],[9E+09,9E+09,9E+09,9E+09,9E+09,9E+09]];
    CONST robtarget Target_2930_2:=[[83.906,61.285,0],[0.119542298,0.027125582,0.159127158,0.979618492],[-1,-1,1,0],[9E+09,9E+09,9E+09,9E+09,9E+09,9E+09]];
    CONST robtarget Target_2940_2:=[[86.008,60.861,0],[0.119542298,0.027125582,0.159127158,0.979618492],[-1,-1,1,0],[9E+09,9E+09,9E+09,9E+09,9E+09,9E+09]];
    CONST robtarget Target_2950_2:=[[87.5,60.861,0],[0.119542298,0.027125582,0.159127158,0.979618492],[-1,-1,1,0],[9E+09,9E+09,9E+09,9E+09,9E+09,9E+09]];
    CONST robtarget Target_2960_2:=[[88.991,60.861,0],[0.119542298,0.027125582,0.159127158,0.979618492],[-1,-1,1,0],[9E+09,9E+09,9E+09,9E+09,9E+09,9E+09]];
    CONST robtarget Target_2970_2:=[[88.991,64.545,0],[0.119542298,0.027125582,0.159127158,0.979618492],[-1,-1,1,0],[9E+09,9E+09,9E+09,9E+09,9E+09,9E+09]];
    CONST robtarget Target_2980_2:=[[88.991,64.545,-10],[0.119542298,0.027125582,0.159127158,0.979618492],[-1,-1,1,0],[9E+09,9E+09,9E+09,9E+09,9E+09,9E+09]];
    CONST robtarget Target_2990_2:=[[73.457,75.499,-10],[0.119542298,0.027125582,0.159127158,0.979618492],[-1,-1,1,0],[9E+09,9E+09,9E+09,9E+09,9E+09,9E+09]];
    CONST robtarget Target_3000_2:=[[73.457,75.499,0],[0.119542298,0.027125582,0.159127158,0.979618492],[-1,-1,1,0],[9E+09,9E+09,9E+09,9E+09,9E+09,9E+09]];
    CONST robtarget Target_3010_2:=[[65.258,75.499,0],[0.119542298,0.027125582,0.159127158,0.979618492],[-1,-1,1,0],[9E+09,9E+09,9E+09,9E+09,9E+09,9E+09]];
    CONST robtarget Target_3020_2:=[[58.665,74.358,0],[0.119542298,0.027125582,0.159127158,0.979618492],[-1,-1,1,0],[9E+09,9E+09,9E+09,9E+09,9E+09,9E+09]];
    CONST robtarget Target_3030_2:=[[56.913,70.446,0],[0.119542298,0.027125582,0.159127158,0.979618492],[-1,-1,1,0],[9E+09,9E+09,9E+09,9E+09,9E+09,9E+09]];
    CONST robtarget Target_3040_2:=[[57.785,67.324,0],[0.119542298,0.027125582,0.159127158,0.979618492],[-1,-1,1,0],[9E+09,9E+09,9E+09,9E+09,9E+09,9E+09]];
    CONST robtarget Target_3050_2:=[[60.613,65.474,0],[0.119542298,0.027125582,0.159127158,0.979618492],[-1,-1,1,0],[9E+09,9E+09,9E+09,9E+09,9E+09,9E+09]];
    CONST robtarget Target_3060_2:=[[57.736,63.95,0],[0.119542298,0.027125582,0.159127158,0.979618492],[-1,-1,1,0],[9E+09,9E+09,9E+09,9E+09,9E+09,9E+09]];
    CONST robtarget Target_3070_2:=[[56.88,61.024,0],[0.119542298,0.027125582,0.159127158,0.979618492],[-1,-1,1,0],[9E+09,9E+09,9E+09,9E+09,9E+09,9E+09]];
    CONST robtarget Target_3080_2:=[[56.799,58.115,0],[0.119542298,0.027125582,0.159127158,0.979618492],[-1,-1,1,0],[9E+09,9E+09,9E+09,9E+09,9E+09,9E+09]];
    CONST robtarget Target_3090_2:=[[56.424,56.819,0],[0.119542298,0.027125582,0.159127158,0.979618492],[-1,-1,1,0],[9E+09,9E+09,9E+09,9E+09,9E+09,9E+09]];
    CONST robtarget Target_3100_2:=[[61.395,56.819,0],[0.119542298,0.027125582,0.159127158,0.979618492],[-1,-1,1,0],[9E+09,9E+09,9E+09,9E+09,9E+09,9E+09]];
    CONST robtarget Target_3110_2:=[[61.656,58.27,0],[0.119542298,0.027125582,0.159127158,0.979618492],[-1,-1,1,0],[9E+09,9E+09,9E+09,9E+09,9E+09,9E+09]];
    CONST robtarget Target_3120_2:=[[61.656,59.394,0],[0.119542298,0.027125582,0.159127158,0.979618492],[-1,-1,1,0],[9E+09,9E+09,9E+09,9E+09,9E+09,9E+09]];
    CONST robtarget Target_3130_2:=[[61.656,60.519,0],[0.119542298,0.027125582,0.159127158,0.979618492],[-1,-1,1,0],[9E+09,9E+09,9E+09,9E+09,9E+09,9E+09]];
    CONST robtarget Target_3140_2:=[[62.43,62.923,0],[0.119542298,0.027125582,0.159127158,0.979618492],[-1,-1,1,0],[9E+09,9E+09,9E+09,9E+09,9E+09,9E+09]];
    CONST robtarget Target_3150_2:=[[64.737,63.714,0],[0.119542298,0.027125582,0.159127158,0.979618492],[-1,-1,1,0],[9E+09,9E+09,9E+09,9E+09,9E+09,9E+09]];
    CONST robtarget Target_3160_2:=[[68.486,63.714,0],[0.119542298,0.027125582,0.159127158,0.979618492],[-1,-1,1,0],[9E+09,9E+09,9E+09,9E+09,9E+09,9E+09]];
    CONST robtarget Target_3170_2:=[[68.486,56.819,0],[0.119542298,0.027125582,0.159127158,0.979618492],[-1,-1,1,0],[9E+09,9E+09,9E+09,9E+09,9E+09,9E+09]];
    CONST robtarget Target_3180_2:=[[73.457,56.819,0],[0.119542298,0.027125582,0.159127158,0.979618492],[-1,-1,1,0],[9E+09,9E+09,9E+09,9E+09,9E+09,9E+09]];
    CONST robtarget Target_3190_2:=[[73.457,75.499,0],[0.119542298,0.027125582,0.159127158,0.979618492],[-1,-1,1,0],[9E+09,9E+09,9E+09,9E+09,9E+09,9E+09]];
    CONST robtarget Target_3200_2:=[[73.457,75.499,-10],[0.119542298,0.027125582,0.159127158,0.979618492],[-1,-1,1,0],[9E+09,9E+09,9E+09,9E+09,9E+09,9E+09]];
    CONST robtarget Target_3210_2:=[[67.801,71.342,-10],[0.119542298,0.027125582,0.159127158,0.979618492],[-1,-1,1,0],[9E+09,9E+09,9E+09,9E+09,9E+09,9E+09]];
    CONST robtarget Target_3220_2:=[[67.801,71.342,0],[0.119542298,0.027125582,0.159127158,0.979618492],[-1,-1,1,0],[9E+09,9E+09,9E+09,9E+09,9E+09,9E+09]];
    CONST robtarget Target_3230_2:=[[65.047,71.342,0],[0.119542298,0.027125582,0.159127158,0.979618492],[-1,-1,1,0],[9E+09,9E+09,9E+09,9E+09,9E+09,9E+09]];
    CONST robtarget Target_3240_2:=[[62.74,70.918,0],[0.119542298,0.027125582,0.159127158,0.979618492],[-1,-1,1,0],[9E+09,9E+09,9E+09,9E+09,9E+09,9E+09]];
    CONST robtarget Target_3250_2:=[[62.178,69.451,0],[0.119542298,0.027125582,0.159127158,0.979618492],[-1,-1,1,0],[9E+09,9E+09,9E+09,9E+09,9E+09,9E+09]];
    CONST robtarget Target_3260_2:=[[62.756,68.017,0],[0.119542298,0.027125582,0.159127158,0.979618492],[-1,-1,1,0],[9E+09,9E+09,9E+09,9E+09,9E+09,9E+09]];
    CONST robtarget Target_3270_2:=[[64.884,67.593,0],[0.119542298,0.027125582,0.159127158,0.979618492],[-1,-1,1,0],[9E+09,9E+09,9E+09,9E+09,9E+09,9E+09]];
    CONST robtarget Target_3280_2:=[[67.801,67.593,0],[0.119542298,0.027125582,0.159127158,0.979618492],[-1,-1,1,0],[9E+09,9E+09,9E+09,9E+09,9E+09,9E+09]];
    CONST robtarget Target_3290_2:=[[67.801,71.342,0],[0.119542298,0.027125582,0.159127158,0.979618492],[-1,-1,1,0],[9E+09,9E+09,9E+09,9E+09,9E+09,9E+09]];
    CONST robtarget Target_3300_2:=[[67.801,71.342,-10],[0.119542298,0.027125582,0.159127158,0.979618492],[-1,-1,1,0],[9E+09,9E+09,9E+09,9E+09,9E+09,9E+09]];
    CONST robtarget Target_3310_2:=[[52.121,75.499,-10],[0.119542298,0.027125582,0.159127158,0.979618492],[-1,-1,1,0],[9E+09,9E+09,9E+09,9E+09,9E+09,9E+09]];
    CONST robtarget Target_3320_2:=[[52.121,75.499,0],[0.119542298,0.027125582,0.159127158,0.979618492],[-1,-1,1,0],[9E+09,9E+09,9E+09,9E+09,9E+09,9E+09]];
    CONST robtarget Target_3330_2:=[[46.954,75.499,0],[0.119542298,0.027125582,0.159127158,0.979618492],[-1,-1,1,0],[9E+09,9E+09,9E+09,9E+09,9E+09,9E+09]];
    CONST robtarget Target_3340_2:=[[46.954,56.819,0],[0.119542298,0.027125582,0.159127158,0.979618492],[-1,-1,1,0],[9E+09,9E+09,9E+09,9E+09,9E+09,9E+09]];
    CONST robtarget Target_3350_2:=[[52.121,56.819,0],[0.119542298,0.027125582,0.159127158,0.979618492],[-1,-1,1,0],[9E+09,9E+09,9E+09,9E+09,9E+09,9E+09]];
    CONST robtarget Target_3360_2:=[[52.121,75.499,0],[0.119542298,0.027125582,0.159127158,0.979618492],[-1,-1,1,0],[9E+09,9E+09,9E+09,9E+09,9E+09,9E+09]];
    CONST robtarget Target_3370_2:=[[52.121,75.499,-10],[0.119542298,0.027125582,0.159127158,0.979618492],[-1,-1,1,0],[9E+09,9E+09,9E+09,9E+09,9E+09,9E+09]];
    CONST robtarget Target_3380_2:=[[41.672,75.499,-10],[0.119542298,0.027125582,0.159127158,0.979618492],[-1,-1,1,0],[9E+09,9E+09,9E+09,9E+09,9E+09,9E+09]];
    CONST robtarget Target_3390_2:=[[41.672,75.499,0],[0.119542298,0.027125582,0.159127158,0.979618492],[-1,-1,1,0],[9E+09,9E+09,9E+09,9E+09,9E+09,9E+09]];
    CONST robtarget Target_3400_2:=[[27.051,75.499,0],[0.119542298,0.027125582,0.159127158,0.979618492],[-1,-1,1,0],[9E+09,9E+09,9E+09,9E+09,9E+09,9E+09]];
    CONST robtarget Target_3410_2:=[[27.051,72.027,0],[0.119542298,0.027125582,0.159127158,0.979618492],[-1,-1,1,0],[9E+09,9E+09,9E+09,9E+09,9E+09,9E+09]];
    CONST robtarget Target_3420_2:=[[36.62,72.027,0],[0.119542298,0.027125582,0.159127158,0.979618492],[-1,-1,1,0],[9E+09,9E+09,9E+09,9E+09,9E+09,9E+09]];
    CONST robtarget Target_3430_2:=[[36.62,68.099,0],[0.119542298,0.027125582,0.159127158,0.979618492],[-1,-1,1,0],[9E+09,9E+09,9E+09,9E+09,9E+09,9E+09]];
    CONST robtarget Target_3440_2:=[[28.535,68.099,0],[0.119542298,0.027125582,0.159127158,0.979618492],[-1,-1,1,0],[9E+09,9E+09,9E+09,9E+09,9E+09,9E+09]];
    CONST robtarget Target_3450_2:=[[28.535,64.773,0],[0.119542298,0.027125582,0.159127158,0.979618492],[-1,-1,1,0],[9E+09,9E+09,9E+09,9E+09,9E+09,9E+09]];
    CONST robtarget Target_3460_2:=[[36.62,64.773,0],[0.119542298,0.027125582,0.159127158,0.979618492],[-1,-1,1,0],[9E+09,9E+09,9E+09,9E+09,9E+09,9E+09]];
    CONST robtarget Target_3470_2:=[[36.62,60.372,0],[0.119542298,0.027125582,0.159127158,0.979618492],[-1,-1,1,0],[9E+09,9E+09,9E+09,9E+09,9E+09,9E+09]];
    CONST robtarget Target_3480_2:=[[26.677,60.372,0],[0.119542298,0.027125582,0.159127158,0.979618492],[-1,-1,1,0],[9E+09,9E+09,9E+09,9E+09,9E+09,9E+09]];
    CONST robtarget Target_3490_2:=[[26.677,56.819,0],[0.119542298,0.027125582,0.159127158,0.979618492],[-1,-1,1,0],[9E+09,9E+09,9E+09,9E+09,9E+09,9E+09]];
    CONST robtarget Target_3500_2:=[[41.672,56.819,0],[0.119542298,0.027125582,0.159127158,0.979618492],[-1,-1,1,0],[9E+09,9E+09,9E+09,9E+09,9E+09,9E+09]];
    CONST robtarget Target_3510_2:=[[41.672,75.499,0],[0.119542298,0.027125582,0.159127158,0.979618492],[-1,-1,1,0],[9E+09,9E+09,9E+09,9E+09,9E+09,9E+09]];
    CONST robtarget Target_3520_2:=[[41.672,75.499,-10],[0.119542298,0.027125582,0.159127158,0.979618492],[-1,-1,1,0],[9E+09,9E+09,9E+09,9E+09,9E+09,9E+09]];
    CONST robtarget Target_3530_2:=[[22.308,75.499,-10],[0.119542298,0.027125582,0.159127158,0.979618492],[-1,-1,1,0],[9E+09,9E+09,9E+09,9E+09,9E+09,9E+09]];
    CONST robtarget Target_3540_2:=[[22.308,75.499,0],[0.119542298,0.027125582,0.159127158,0.979618492],[-1,-1,1,0],[9E+09,9E+09,9E+09,9E+09,9E+09,9E+09]];
    CONST robtarget Target_3550_2:=[[17.255,75.499,0],[0.119542298,0.027125582,0.159127158,0.979618492],[-1,-1,1,0],[9E+09,9E+09,9E+09,9E+09,9E+09,9E+09]];
    CONST robtarget Target_3560_2:=[[17.255,60.829,0],[0.119542298,0.027125582,0.159127158,0.979618492],[-1,-1,1,0],[9E+09,9E+09,9E+09,9E+09,9E+09,9E+09]];
    CONST robtarget Target_3570_2:=[[8.518,60.829,0],[0.119542298,0.027125582,0.159127158,0.979618492],[-1,-1,1,0],[9E+09,9E+09,9E+09,9E+09,9E+09,9E+09]];
    CONST robtarget Target_3580_2:=[[8.518,56.819,0],[0.119542298,0.027125582,0.159127158,0.979618492],[-1,-1,1,0],[9E+09,9E+09,9E+09,9E+09,9E+09,9E+09]];
    CONST robtarget Target_3590_2:=[[22.308,56.819,0],[0.119542298,0.027125582,0.159127158,0.979618492],[-1,-1,1,0],[9E+09,9E+09,9E+09,9E+09,9E+09,9E+09]];
    CONST robtarget Target_3600_2:=[[22.308,75.499,0],[0.119542298,0.027125582,0.159127158,0.979618492],[-1,-1,1,0],[9E+09,9E+09,9E+09,9E+09,9E+09,9E+09]];
    CONST robtarget Target_3610_2:=[[22.308,75.499,-10],[0.119542298,0.027125582,0.159127158,0.979618492],[-2,0,1,0],[9E+09,9E+09,9E+09,9E+09,9E+09,9E+09]];
    CONST robtarget Target_3620_2:=[[94.194,38.558,-10],[0.119542298,0.027125582,0.159127158,0.979618492],[-1,-1,1,0],[9E+09,9E+09,9E+09,9E+09,9E+09,9E+09]];
    CONST robtarget Target_3630_2:=[[94.194,38.558,0],[0.119542298,0.027125582,0.159127158,0.979618492],[-1,-1,1,0],[9E+09,9E+09,9E+09,9E+09,9E+09,9E+09]];
    CONST robtarget Target_3640_2:=[[75.235,49.668,0],[0.119542298,0.027125582,0.159127158,0.979618492],[-1,-1,1,0],[9E+09,9E+09,9E+09,9E+09,9E+09,9E+09]];
    CONST robtarget Target_3650_2:=[[56.071,38.286,0],[0.119542298,0.027125582,0.159127158,0.979618492],[-1,-1,1,0],[9E+09,9E+09,9E+09,9E+09,9E+09,9E+09]];
    CONST robtarget Target_3660_2:=[[56.071,16.422,0],[0.119542298,0.027125582,0.159127158,0.979618492],[-1,-1,1,0],[9E+09,9E+09,9E+09,9E+09,9E+09,9E+09]];
    CONST robtarget Target_3670_2:=[[75.083,5.281,0],[0.119542298,0.027125582,0.159127158,0.979618492],[-1,-1,1,0],[9E+09,9E+09,9E+09,9E+09,9E+09,9E+09]];
    CONST robtarget Target_3680_2:=[[94.194,16.631,0],[0.119542298,0.027125582,0.159127158,0.979618492],[-1,-1,1,0],[9E+09,9E+09,9E+09,9E+09,9E+09,9E+09]];
    CONST robtarget Target_3690_2:=[[94.194,38.558,0],[0.119542298,0.027125582,0.159127158,0.979618492],[-1,-1,1,0],[9E+09,9E+09,9E+09,9E+09,9E+09,9E+09]];
    CONST robtarget Target_3700_2:=[[94.194,38.558,-10],[0.119542298,0.027125582,0.159127158,0.979618492],[-1,-1,1,0],[9E+09,9E+09,9E+09,9E+09,9E+09,9E+09]];
    CONST robtarget Target_3710_2:=[[89.358,36.21,-10],[0.119542298,0.027125582,0.159127158,0.979618492],[-1,-1,1,0],[9E+09,9E+09,9E+09,9E+09,9E+09,9E+09]];
    CONST robtarget Target_3720_2:=[[89.358,36.21,0],[0.119542298,0.027125582,0.159127158,0.979618492],[-1,-1,1,0],[9E+09,9E+09,9E+09,9E+09,9E+09,9E+09]];
    CONST robtarget Target_3730_2:=[[75.235,44.113,0],[0.119542298,0.027125582,0.159127158,0.979618492],[-1,-1,1,0],[9E+09,9E+09,9E+09,9E+09,9E+09,9E+09]];
    CONST robtarget Target_3740_2:=[[72.307,41.696,0],[0.119542298,0.027125582,0.159127158,0.979618492],[-1,-1,1,0],[9E+09,9E+09,9E+09,9E+09,9E+09,9E+09]];
    CONST robtarget Target_3750_2:=[[70.636,38.286,0],[0.119542298,0.027125582,0.159127158,0.979618492],[-1,-1,1,0],[9E+09,9E+09,9E+09,9E+09,9E+09,9E+09]];
    CONST robtarget Target_3760_2:=[[81.246,14.208,0],[0.119542298,0.027125582,0.159127158,0.979618492],[-1,-1,1,0],[9E+09,9E+09,9E+09,9E+09,9E+09,9E+09]];
    CONST robtarget Target_3770_2:=[[85.302,16.617,0],[0.119542298,0.027125582,0.159127158,0.979618492],[-1,-1,1,0],[9E+09,9E+09,9E+09,9E+09,9E+09,9E+09]];
    CONST robtarget Target_3780_2:=[[89.358,19.026,0],[0.119542298,0.027125582,0.159127158,0.979618492],[-1,-1,1,0],[9E+09,9E+09,9E+09,9E+09,9E+09,9E+09]];
    CONST robtarget Target_3790_2:=[[89.358,36.21,0],[0.119542298,0.027125582,0.159127158,0.979618492],[-1,-1,1,0],[9E+09,9E+09,9E+09,9E+09,9E+09,9E+09]];
    CONST robtarget Target_3800_2:=[[89.358,36.21,-10],[0.119542298,0.027125582,0.159127158,0.979618492],[-1,-1,1,0],[9E+09,9E+09,9E+09,9E+09,9E+09,9E+09]];
    CONST robtarget Target_3810_2:=[[68.77,34.464,-10],[0.119542298,0.027125582,0.159127158,0.979618492],[-1,-1,1,0],[9E+09,9E+09,9E+09,9E+09,9E+09,9E+09]];
    CONST robtarget Target_3820_2:=[[68.77,34.464,0],[0.119542298,0.027125582,0.159127158,0.979618492],[-1,-1,1,0],[9E+09,9E+09,9E+09,9E+09,9E+09,9E+09]];
    CONST robtarget Target_3830_2:=[[62.422,17.88,0],[0.119542298,0.027125582,0.159127158,0.979618492],[-1,-1,1,0],[9E+09,9E+09,9E+09,9E+09,9E+09,9E+09]];
    CONST robtarget Target_3840_2:=[[74.993,10.536,0],[0.119542298,0.027125582,0.159127158,0.979618492],[-1,-1,1,0],[9E+09,9E+09,9E+09,9E+09,9E+09,9E+09]];
    CONST robtarget Target_3850_2:=[[77.735,12.123,0],[0.119542298,0.027125582,0.159127158,0.979618492],[-1,-1,1,0],[9E+09,9E+09,9E+09,9E+09,9E+09,9E+09]];
    CONST robtarget Target_3860_2:=[[68.77,34.464,0],[0.119542298,0.027125582,0.159127158,0.979618492],[-1,-1,1,0],[9E+09,9E+09,9E+09,9E+09,9E+09,9E+09]];
    CONST robtarget Target_3870_2:=[[68.77,34.464,-10],[0.119542298,0.027125582,0.159127158,0.979618492],[-1,-1,1,0],[9E+09,9E+09,9E+09,9E+09,9E+09,9E+09]];
    CONST robtarget Target_3880_2:=[[67.293,40.162,-10],[0.119542298,0.027125582,0.159127158,0.979618492],[-1,-1,1,0],[9E+09,9E+09,9E+09,9E+09,9E+09,9E+09]];
    CONST robtarget Target_3890_2:=[[67.293,40.162,0],[0.119542298,0.027125582,0.159127158,0.979618492],[-1,-1,1,0],[9E+09,9E+09,9E+09,9E+09,9E+09,9E+09]];
    CONST robtarget Target_3900_2:=[[60.509,36.21,0],[0.119542298,0.027125582,0.159127158,0.979618492],[-1,-1,1,0],[9E+09,9E+09,9E+09,9E+09,9E+09,9E+09]];
    CONST robtarget Target_3910_2:=[[60.509,24.537,0],[0.119542298,0.027125582,0.159127158,0.979618492],[-1,-1,1,0],[9E+09,9E+09,9E+09,9E+09,9E+09,9E+09]];
    CONST robtarget Target_3920_2:=[[67.293,40.162,0],[0.119542298,0.027125582,0.159127158,0.979618492],[-1,-1,1,0],[9E+09,9E+09,9E+09,9E+09,9E+09,9E+09]];
    CONST robtarget Target_3930_2:=[[67.472477576,40.059752487,-14.996049097],[0.119542298,0.027125582,0.159127158,0.979618492],[-2,-1,1,0],[9E+09,9E+09,9E+09,9E+09,9E+09,9E+09]];
    CONST robtarget Target_3940_2:=[[68.00538685,-48.442633556,-13.16160056],[0.119542298,0.027125582,0.159127158,0.979618492],[-2,-1,1,0],[9E+09,9E+09,9E+09,9E+09,9E+09,9E+09]];
    !***********************************************************
    !
    ! M?dulo:  Module1
    !
    ! Descripción:
    !   <Introduzca la descripción aquí>
    !
    ! Autor: Gabriel Bojaca
    !
    ! Versión: 1.0
    !
    !***********************************************************


    !***********************************************************
    !
    ! Procedimiento Main
    !
    !   Este es el punto de entrada de su programa
    !
    !***********************************************************
    PROC main()

        TPErase;
        TPWrite "INICIO PROGRAMA";
        TPWrite "APAGADO BANDA TRANASPORTADORA";
        Reset Conveyor_FWD;
        Reset DO_02;

        WHILE TRUE DO
            IF DI_01 = 1 AND DI_02 = 0 THEN
                TPWrite "ENCIENDE BANDA TRANASPORTADORA";
                Set Conveyor_FWD;
                WaitTime 3;
                TPWrite "APAGADO BANDA TRANASPORTADORA";
                Reset Conveyor_FWD;
                TPWrite "INICIANDO DECORADO";
                Set DO_02;
                MoveAbsJ SINGBREAK, v500, z1, Marcador;
                ANICOLAS;
                TPWrite "DECORADO COMPLETADO 1/4";
                BCAMILO;
                TPWrite "DECORADO COMPLETADO 2/4";
                CGABRIEL;
                TPWrite "DECORADO COMPLETADO 3/4";
                DKYMA;
                TPWrite "DECORADO FINALIZADO";
                Homming;
                WaitTime 3;
                TPWrite "ENCENDIDO BANDA TRANASPORTADORA";
                Set Conveyor_FWD;
                WaitTime 5;
                TPWrite "APAGADO BANDA TRANASPORTADORA";
                Reset Conveyor_FWD;

            ELSEIF DI_01 = 0 AND DI_02=1 THEN
                TPWrite "RUTINA CAMBIO DE HERRAMIENTA";
                Homming;
                MoveAbsJ CHANGETOOL, v500, z5, Marcador;
                Reset DO_02;
                TPWrite "PELIGRO";
                TPWrite "OPERARIO CERCA A HERRAMIENTA";
                TPWrite "PRESIONE LOS DOS BOTONES PARA CONTINUAR EL PROGRAMA";
                WaitDI DI_01,1;
                WaitDI DI_02,1;
            TPWrite "REANUDANDO PROGRAMA";
            WaitTime 5;
            MoveAbsJ home0, v500, fine, Marcador;
            ELSEIF DI_01 = 0 AND DI_02=0 THEN
                TPWrite "ESPERANDO INSTRUCCIÓNES";
                WaitTime 1;
            ELSEIF DI_01 = 1 AND DI_02=1 THEN
                TPWrite "ERROR";
                TPWrite "NO DEBE PRESIONAR AMBAS ENTRADAS AL TIEMPO";
                WaitTime 1;
            ENDIF

        ENDWHILE




        !WaitDI DI_02,1; !Rutina de prueba de Homming
        !Homming;









    ENDPROC
    PROC ANICOLAS()
        MoveJ HOME,v100,z1,Marcador\WObj:=Pastel;
        MoveL Aproximacion,v100,z1,Marcador\WObj:=Pastel;
        MoveL Target_10,v100,z1,Marcador\WObj:=Pastel;
        MoveL Target_20,v100,z1,Marcador\WObj:=Pastel;
        MoveL Target_30,v100,z1,Marcador\WObj:=Pastel;
        MoveL Target_40,v100,z1,Marcador\WObj:=Pastel;
        MoveL Target_50,v100,z1,Marcador\WObj:=Pastel;
        MoveL Target_60,v100,z1,Marcador\WObj:=Pastel;
        MoveL Target_70,v100,z1,Marcador\WObj:=Pastel;
        MoveL Target_80,v100,z1,Marcador\WObj:=Pastel;
        MoveL Target_90,v100,z1,Marcador\WObj:=Pastel;
        MoveL Target_100,v100,z1,Marcador\WObj:=Pastel;
        MoveL Target_110,v100,z1,Marcador\WObj:=Pastel;
        MoveL Target_120,v100,z1,Marcador\WObj:=Pastel;
        MoveL Target_130,v100,z1,Marcador\WObj:=Pastel;
        MoveL Target_140,v100,z1,Marcador\WObj:=Pastel;
        MoveL Target_150,v100,z1,Marcador\WObj:=Pastel;
        MoveL Target_160,v100,z1,Marcador\WObj:=Pastel;
        MoveL Target_170,v100,z1,Marcador\WObj:=Pastel;
        MoveL Target_180,v100,z1,Marcador\WObj:=Pastel;
        MoveL Target_190,v100,z1,Marcador\WObj:=Pastel;
        MoveL Target_200,v100,z1,Marcador\WObj:=Pastel;
        MoveL Target_210,v100,z1,Marcador\WObj:=Pastel;
        MoveL Target_220,v100,z1,Marcador\WObj:=Pastel;
        MoveL Target_230,v100,z1,Marcador\WObj:=Pastel;
        MoveL Target_240,v100,z1,Marcador\WObj:=Pastel;
        MoveL Target_250,v100,z1,Marcador\WObj:=Pastel;
        MoveL Target_260,v100,z1,Marcador\WObj:=Pastel;
        MoveL Target_270,v100,z1,Marcador\WObj:=Pastel;
        MoveL Target_280,v100,z1,Marcador\WObj:=Pastel;
        MoveL Target_290,v100,z1,Marcador\WObj:=Pastel;
        MoveL Target_300,v100,z1,Marcador\WObj:=Pastel;
        MoveL Target_310,v100,z1,Marcador\WObj:=Pastel;
        MoveL Target_320,v100,z1,Marcador\WObj:=Pastel;
        MoveL Target_330,v100,z1,Marcador\WObj:=Pastel;
        MoveL Target_340,v100,z1,Marcador\WObj:=Pastel;
        MoveL Target_350,v100,z1,Marcador\WObj:=Pastel;
        MoveL Target_360,v100,z1,Marcador\WObj:=Pastel;
        MoveL Target_370,v100,z1,Marcador\WObj:=Pastel;
        MoveL Target_380,v100,z1,Marcador\WObj:=Pastel;
        MoveL Target_390,v100,z1,Marcador\WObj:=Pastel;
        MoveL Target_400,v100,z1,Marcador\WObj:=Pastel;
        MoveL Target_410,v100,z1,Marcador\WObj:=Pastel;
        MoveL Target_420,v100,z1,Marcador\WObj:=Pastel;
        MoveL Target_430,v100,z1,Marcador\WObj:=Pastel;
        MoveL Target_440,v100,z1,Marcador\WObj:=Pastel;
        MoveL Target_450,v100,z1,Marcador\WObj:=Pastel;
        MoveL Target_460,v100,z1,Marcador\WObj:=Pastel;
        MoveL Target_470,v100,z1,Marcador\WObj:=Pastel;
        MoveL Target_480,v100,z1,Marcador\WObj:=Pastel;
        MoveL Target_490,v100,z1,Marcador\WObj:=Pastel;
        MoveL Target_500,v100,z1,Marcador\WObj:=Pastel;
        MoveL Target_510,v100,z1,Marcador\WObj:=Pastel;
        MoveL Target_520,v100,z1,Marcador\WObj:=Pastel;
        MoveL Target_530,v100,z1,Marcador\WObj:=Pastel;
        MoveL Target_540,v100,z1,Marcador\WObj:=Pastel;
        MoveL Target_550,v100,z1,Marcador\WObj:=Pastel;
        MoveL Target_560,v100,z1,Marcador\WObj:=Pastel;
        MoveL Target_570,v100,z1,Marcador\WObj:=Pastel;
        MoveL Target_580,v100,z1,Marcador\WObj:=Pastel;
        MoveL Target_590,v100,z1,Marcador\WObj:=Pastel;
        MoveL Target_600,v100,z1,Marcador\WObj:=Pastel;
        MoveL Target_610,v100,z1,Marcador\WObj:=Pastel;
        MoveL Target_620,v100,z1,Marcador\WObj:=Pastel;
        MoveL Target_630,v100,z1,Marcador\WObj:=Pastel;
        MoveL Target_640,v100,z1,Marcador\WObj:=Pastel;
        MoveL Target_650,v100,z1,Marcador\WObj:=Pastel;
        MoveL Target_660,v100,z1,Marcador\WObj:=Pastel;
        MoveL Target_670,v100,z1,Marcador\WObj:=Pastel;
        MoveL Target_680,v100,z1,Marcador\WObj:=Pastel;
        MoveL Target_690,v100,z1,Marcador\WObj:=Pastel;
        MoveL Target_700,v100,z1,Marcador\WObj:=Pastel;
        MoveL Target_710,v100,z1,Marcador\WObj:=Pastel;
        MoveL Target_720,v100,z1,Marcador\WObj:=Pastel;
        MoveL Target_730,v100,z1,Marcador\WObj:=Pastel;
        MoveL Target_740,v100,z1,Marcador\WObj:=Pastel;
        MoveL Target_750,v100,z1,Marcador\WObj:=Pastel;
        MoveL Target_760,v100,z1,Marcador\WObj:=Pastel;
        MoveL Target_770,v100,z1,Marcador\WObj:=Pastel;
        MoveL Target_780,v100,z1,Marcador\WObj:=Pastel;
        MoveL Target_790,v100,z1,Marcador\WObj:=Pastel;
        MoveL Target_800,v100,z1,Marcador\WObj:=Pastel;
        MoveL Target_810,v100,z1,Marcador\WObj:=Pastel;
        MoveL Target_820,v100,z1,Marcador\WObj:=Pastel;
        MoveL Target_830,v100,z1,Marcador\WObj:=Pastel;
        MoveL Target_840,v100,z1,Marcador\WObj:=Pastel;
        MoveL Target_850,v100,z1,Marcador\WObj:=Pastel;
        MoveL Target_860,v100,z1,Marcador\WObj:=Pastel;
        MoveL Target_870,v100,z1,Marcador\WObj:=Pastel;
        MoveL Target_880,v100,z1,Marcador\WObj:=Pastel;
        MoveL Target_890,v100,z1,Marcador\WObj:=Pastel;
        MoveL Target_900,v100,z1,Marcador\WObj:=Pastel;
        MoveL Target_910,v100,z1,Marcador\WObj:=Pastel;
        MoveL Target_920,v100,z1,Marcador\WObj:=Pastel;
        MoveL Target_930,v100,z1,Marcador\WObj:=Pastel;
        MoveL Target_940,v100,z1,Marcador\WObj:=Pastel;
        MoveL Target_950,v100,z1,Marcador\WObj:=Pastel;
        MoveL Target_960,v100,z1,Marcador\WObj:=Pastel;
        MoveL Target_970,v100,z1,Marcador\WObj:=Pastel;
        MoveL Target_980,v100,z1,Marcador\WObj:=Pastel;
        MoveL Target_990,v100,z1,Marcador\WObj:=Pastel;
        MoveL Target_1000,v100,z1,Marcador\WObj:=Pastel;
        MoveL Target_1010,v100,z1,Marcador\WObj:=Pastel;
        MoveL Target_1020,v100,z1,Marcador\WObj:=Pastel;
        MoveL Target_1030,v100,z1,Marcador\WObj:=Pastel;
        MoveL Target_1040,v100,z1,Marcador\WObj:=Pastel;
        MoveL Target_1050,v100,z1,Marcador\WObj:=Pastel;
        MoveL Target_1060,v100,z1,Marcador\WObj:=Pastel;
        MoveL Target_1070,v100,z1,Marcador\WObj:=Pastel;
        MoveL Target_1080,v100,z1,Marcador\WObj:=Pastel;
        MoveL Target_1090,v100,z1,Marcador\WObj:=Pastel;
        MoveL Target_1100,v100,z1,Marcador\WObj:=Pastel;
        MoveL Target_1110,v100,z1,Marcador\WObj:=Pastel;
        MoveL Target_1120,v100,z1,Marcador\WObj:=Pastel;
        MoveL Target_1130,v100,z1,Marcador\WObj:=Pastel;
        MoveL Target_1140,v100,z1,Marcador\WObj:=Pastel;
        MoveL Target_1150,v100,z1,Marcador\WObj:=Pastel;
        MoveL Target_1160,v100,z1,Marcador\WObj:=Pastel;
        MoveL Target_1170,v100,z1,Marcador\WObj:=Pastel;
        MoveL Target_1180,v100,z1,Marcador\WObj:=Pastel;
        MoveL Target_1190,v100,z1,Marcador\WObj:=Pastel;
        MoveL Target_1200,v100,z1,Marcador\WObj:=Pastel;
    ENDPROC
    PROC BCAMILO()
        MoveL Target_1210,v100,z1,Marcador\WObj:=Pastel;
        MoveL Target_1220,v100,z1,Marcador\WObj:=Pastel;
        MoveL Target_1230,v100,z1,Marcador\WObj:=Pastel;
        MoveL Target_1240,v100,z1,Marcador\WObj:=Pastel;
        MoveL Target_1250,v100,z1,Marcador\WObj:=Pastel;
        MoveL Target_1260,v100,z1,Marcador\WObj:=Pastel;
        MoveL Target_1270,v100,z1,Marcador\WObj:=Pastel;
        MoveL Target_1280,v100,z1,Marcador\WObj:=Pastel;
        MoveL Target_1290,v100,z1,Marcador\WObj:=Pastel;
        MoveL Target_1300,v100,z1,Marcador\WObj:=Pastel;
        MoveL Target_1310,v100,z1,Marcador\WObj:=Pastel;
        MoveL Target_1320,v100,z1,Marcador\WObj:=Pastel;
        MoveL Target_1330,v100,z1,Marcador\WObj:=Pastel;
        MoveL Target_1340,v100,z1,Marcador\WObj:=Pastel;
        MoveL Target_1350,v100,z1,Marcador\WObj:=Pastel;
        MoveL Target_1360,v100,z1,Marcador\WObj:=Pastel;
        MoveL Target_1370,v100,z1,Marcador\WObj:=Pastel;
        MoveL Target_1380,v100,z1,Marcador\WObj:=Pastel;
        MoveL Target_1390,v100,z1,Marcador\WObj:=Pastel;
        MoveL Target_1400,v100,z1,Marcador\WObj:=Pastel;
        MoveL Target_1410,v100,z1,Marcador\WObj:=Pastel;
        MoveL Target_1420,v100,z1,Marcador\WObj:=Pastel;
        MoveL Target_1430,v100,z1,Marcador\WObj:=Pastel;
        MoveL Target_1440,v100,z1,Marcador\WObj:=Pastel;
        MoveL Target_1450,v100,z1,Marcador\WObj:=Pastel;
        MoveL Target_1460,v100,z1,Marcador\WObj:=Pastel;
        MoveL Target_1470,v100,z1,Marcador\WObj:=Pastel;
        MoveL Target_1480,v100,z1,Marcador\WObj:=Pastel;
        MoveL Target_1490,v100,z1,Marcador\WObj:=Pastel;
        MoveL Target_1500,v100,z1,Marcador\WObj:=Pastel;
        MoveL Target_1510,v100,z1,Marcador\WObj:=Pastel;
        MoveL Target_1520,v100,z1,Marcador\WObj:=Pastel;
        MoveL Target_1530,v100,z1,Marcador\WObj:=Pastel;
        MoveL Target_1540,v100,z1,Marcador\WObj:=Pastel;
        MoveL Target_1550,v100,z1,Marcador\WObj:=Pastel;
        MoveL Target_1560,v100,z1,Marcador\WObj:=Pastel;
        MoveL Target_1570,v100,z1,Marcador\WObj:=Pastel;
        MoveL Target_1580,v100,z1,Marcador\WObj:=Pastel;
        MoveL Target_1590,v100,z1,Marcador\WObj:=Pastel;
        MoveL Target_1600,v100,z1,Marcador\WObj:=Pastel;
        MoveL Target_1610,v100,z1,Marcador\WObj:=Pastel;
        MoveL Target_1620,v100,z1,Marcador\WObj:=Pastel;
        MoveL Target_1630,v100,z1,Marcador\WObj:=Pastel;
        MoveL Target_1640,v100,z1,Marcador\WObj:=Pastel;
        MoveL Target_1650,v100,z1,Marcador\WObj:=Pastel;
        MoveL Target_1660,v100,z1,Marcador\WObj:=Pastel;
        MoveL Target_1670,v100,z1,Marcador\WObj:=Pastel;
        MoveL Target_1680,v100,z1,Marcador\WObj:=Pastel;
        MoveL Target_1690,v100,z1,Marcador\WObj:=Pastel;
        MoveL Target_1700,v100,z1,Marcador\WObj:=Pastel;
        MoveL Target_1710,v100,z1,Marcador\WObj:=Pastel;
        MoveL Target_1720,v100,z1,Marcador\WObj:=Pastel;
        MoveL Target_1730,v100,z1,Marcador\WObj:=Pastel;
        MoveL Target_1740,v100,z1,Marcador\WObj:=Pastel;
        MoveL Target_1750,v100,z1,Marcador\WObj:=Pastel;
        MoveL Target_1760,v100,z1,Marcador\WObj:=Pastel;
        MoveL Target_1770,v100,z1,Marcador\WObj:=Pastel;
        MoveL Target_1780,v100,z1,Marcador\WObj:=Pastel;
        MoveL Target_1790,v100,z1,Marcador\WObj:=Pastel;
        MoveL Target_1800,v100,z1,Marcador\WObj:=Pastel;
        MoveL Target_1810,v100,z1,Marcador\WObj:=Pastel;
        MoveL Target_1820,v100,z1,Marcador\WObj:=Pastel;
        MoveL Target_1830,v100,z1,Marcador\WObj:=Pastel;
        MoveL Target_1840,v100,z1,Marcador\WObj:=Pastel;
        MoveL Target_1850,v100,z1,Marcador\WObj:=Pastel;
        MoveL Target_1860,v100,z1,Marcador\WObj:=Pastel;
        MoveL Target_1870,v100,z1,Marcador\WObj:=Pastel;
        MoveL Target_1880,v100,z1,Marcador\WObj:=Pastel;
        MoveL Target_1890,v100,z1,Marcador\WObj:=Pastel;
        MoveL Target_1900,v100,z1,Marcador\WObj:=Pastel;
        MoveL Target_1910,v100,z1,Marcador\WObj:=Pastel;
        MoveL Target_1920,v100,z1,Marcador\WObj:=Pastel;
        MoveL Target_1930,v100,z1,Marcador\WObj:=Pastel;
        MoveL Target_1940,v100,z1,Marcador\WObj:=Pastel;
        MoveL Target_1950,v100,z1,Marcador\WObj:=Pastel;
        MoveL Target_1960,v100,z1,Marcador\WObj:=Pastel;
        MoveL Target_1970,v100,z1,Marcador\WObj:=Pastel;
        MoveL Target_1980,v100,z1,Marcador\WObj:=Pastel;
        MoveL Target_1990,v100,z1,Marcador\WObj:=Pastel;
        MoveL Target_2000,v100,z1,Marcador\WObj:=Pastel;
        MoveL Target_2010,v100,z1,Marcador\WObj:=Pastel;
        MoveL Target_2020,v100,z1,Marcador\WObj:=Pastel;
        MoveL Target_2030,v100,z1,Marcador\WObj:=Pastel;
        MoveL Target_2040,v100,z1,Marcador\WObj:=Pastel;
        MoveL Target_2050,v100,z1,Marcador\WObj:=Pastel;
        MoveL Target_2060,v100,z1,Marcador\WObj:=Pastel;
        MoveL Target_2070,v100,z1,Marcador\WObj:=Pastel;
        MoveL Target_2080,v100,z1,Marcador\WObj:=Pastel;
        MoveL Target_2090,v100,z1,Marcador\WObj:=Pastel;
        MoveL Target_2100,v100,z1,Marcador\WObj:=Pastel;
        MoveL Target_2110,v100,z1,Marcador\WObj:=Pastel;
        MoveL Target_2120,v100,z1,Marcador\WObj:=Pastel;
        MoveL Target_2130,v100,z1,Marcador\WObj:=Pastel;
        MoveL Target_2140,v100,z1,Marcador\WObj:=Pastel;
    ENDPROC
    PROC CGABRIEL()
        MoveL Target_2150,v100,z1,Marcador\WObj:=Pastel;
        MoveL Target_2160,v100,z1,Marcador\WObj:=Pastel;
        MoveL Target_2170,v100,z1,Marcador\WObj:=Pastel;
        MoveL Target_2180,v100,z1,Marcador\WObj:=Pastel;
        MoveL Target_2190,v100,z1,Marcador\WObj:=Pastel;
        MoveL Target_2200,v100,z1,Marcador\WObj:=Pastel;
        MoveL Target_2210,v100,z1,Marcador\WObj:=Pastel;
        MoveL Target_2220,v100,z1,Marcador\WObj:=Pastel;
        MoveL Target_2230,v100,z1,Marcador\WObj:=Pastel;
        MoveL Target_2240,v100,z1,Marcador\WObj:=Pastel;
        MoveL Target_2250,v100,z1,Marcador\WObj:=Pastel;
        MoveL Target_2260,v100,z1,Marcador\WObj:=Pastel;
        MoveL Target_2270,v100,z1,Marcador\WObj:=Pastel;
        MoveL Target_2280,v100,z1,Marcador\WObj:=Pastel;
        MoveL Target_2290,v100,z1,Marcador\WObj:=Pastel;
        MoveL Target_2300,v100,z1,Marcador\WObj:=Pastel;
        MoveL Target_2310,v100,z1,Marcador\WObj:=Pastel;
        MoveL Target_2320,v100,z1,Marcador\WObj:=Pastel;
        MoveL Target_2330,v100,z1,Marcador\WObj:=Pastel;
        MoveL Target_2340,v100,z1,Marcador\WObj:=Pastel;
        MoveL Target_2350,v100,z1,Marcador\WObj:=Pastel;
        MoveL Target_2360,v100,z1,Marcador\WObj:=Pastel;
        MoveL Target_2370,v100,z1,Marcador\WObj:=Pastel;
        MoveL Target_2380,v100,z1,Marcador\WObj:=Pastel;
        MoveL Target_2390,v100,z1,Marcador\WObj:=Pastel;
        MoveL Target_2400,v100,z1,Marcador\WObj:=Pastel;
        MoveL Target_2410,v100,z1,Marcador\WObj:=Pastel;
        MoveL Target_2420,v100,z1,Marcador\WObj:=Pastel;
        MoveL Target_2430,v100,z1,Marcador\WObj:=Pastel;
        MoveL Target_2440,v100,z1,Marcador\WObj:=Pastel;
        MoveL Target_2450,v100,z1,Marcador\WObj:=Pastel;
        MoveL Target_2460,v100,z1,Marcador\WObj:=Pastel;
        MoveL Target_2470,v100,z1,Marcador\WObj:=Pastel;
        MoveL Target_2480,v100,z1,Marcador\WObj:=Pastel;
        MoveL Target_2490,v100,z1,Marcador\WObj:=Pastel;
        MoveL Target_2500,v100,z1,Marcador\WObj:=Pastel;
        MoveL Target_2510,v100,z1,Marcador\WObj:=Pastel;
        MoveL Target_2520,v100,z1,Marcador\WObj:=Pastel;
        MoveL Target_2530,v100,z1,Marcador\WObj:=Pastel;
        MoveL Target_2540,v100,z1,Marcador\WObj:=Pastel;
        MoveL Target_2550,v100,z1,Marcador\WObj:=Pastel;
        MoveL Target_2560,v100,z1,Marcador\WObj:=Pastel;
        MoveL Target_2570,v100,z1,Marcador\WObj:=Pastel;
        MoveL Target_2580,v100,z1,Marcador\WObj:=Pastel;
        MoveL Target_2590,v100,z1,Marcador\WObj:=Pastel;
        MoveL Target_2600,v100,z1,Marcador\WObj:=Pastel;
        MoveL Target_2610,v100,z1,Marcador\WObj:=Pastel;
        MoveL Target_2620,v100,z1,Marcador\WObj:=Pastel;
        MoveL Target_2630,v100,z1,Marcador\WObj:=Pastel;
        MoveL Target_2640,v100,z1,Marcador\WObj:=Pastel;
        MoveL Target_2650,v100,z1,Marcador\WObj:=Pastel;
        MoveL Target_2660,v100,z1,Marcador\WObj:=Pastel;
        MoveL Target_2670,v100,z1,Marcador\WObj:=Pastel;
        MoveL Target_2680,v100,z1,Marcador\WObj:=Pastel;
        MoveL Target_2690,v100,z1,Marcador\WObj:=Pastel;
        MoveL Target_2700,v100,z1,Marcador\WObj:=Pastel;
        MoveL Target_2710,v100,z1,Marcador\WObj:=Pastel;
        MoveL Target_2720,v100,z1,Marcador\WObj:=Pastel;
        MoveL Target_2730,v100,z1,Marcador\WObj:=Pastel;
        MoveL Target_2740,v100,z1,Marcador\WObj:=Pastel;
        MoveL Target_2750,v100,z1,Marcador\WObj:=Pastel;
        MoveL Target_2760,v100,z1,Marcador\WObj:=Pastel;
        MoveL Target_2770,v100,z1,Marcador\WObj:=Pastel;
        MoveL Target_2780,v100,z1,Marcador\WObj:=Pastel;
        MoveL Target_2790,v100,z1,Marcador\WObj:=Pastel;
        MoveL Target_2800,v100,z1,Marcador\WObj:=Pastel;
        MoveL Target_2810,v100,z1,Marcador\WObj:=Pastel;
        MoveL Target_2820,v100,z1,Marcador\WObj:=Pastel;
        MoveL Target_2830,v100,z1,Marcador\WObj:=Pastel;
        MoveL Target_2840,v100,z1,Marcador\WObj:=Pastel;
        MoveL Target_2850,v100,z1,Marcador\WObj:=Pastel;
        MoveL Target_2860,v100,z1,Marcador\WObj:=Pastel;
        MoveL Target_2870,v100,z1,Marcador\WObj:=Pastel;
        MoveL Target_2880,v100,z1,Marcador\WObj:=Pastel;
        MoveL Target_2890,v100,z1,Marcador\WObj:=Pastel;
        MoveL Target_2900,v100,z1,Marcador\WObj:=Pastel;
        MoveL Target_2910,v100,z1,Marcador\WObj:=Pastel;
        MoveL Target_2920,v100,z1,Marcador\WObj:=Pastel;
        MoveL Target_2930,v100,z1,Marcador\WObj:=Pastel;
        MoveL Target_2940,v100,z1,Marcador\WObj:=Pastel;
        MoveL Target_2950,v100,z1,Marcador\WObj:=Pastel;
        MoveL Target_2960,v100,z1,Marcador\WObj:=Pastel;
        MoveL Target_2970,v100,z1,Marcador\WObj:=Pastel;
        MoveL Target_2980,v100,z1,Marcador\WObj:=Pastel;
        MoveL Target_2990,v100,z1,Marcador\WObj:=Pastel;
        MoveL Target_3000,v100,z1,Marcador\WObj:=Pastel;
        MoveL Target_3010,v100,z1,Marcador\WObj:=Pastel;
        MoveL Target_3020,v100,z1,Marcador\WObj:=Pastel;
        MoveL Target_3030,v100,z1,Marcador\WObj:=Pastel;
        MoveL Target_3040,v100,z1,Marcador\WObj:=Pastel;
        MoveL Target_3050,v100,z1,Marcador\WObj:=Pastel;
        MoveL Target_3060,v100,z1,Marcador\WObj:=Pastel;
        MoveL Target_3070,v100,z1,Marcador\WObj:=Pastel;
        MoveL Target_3080,v100,z1,Marcador\WObj:=Pastel;
        MoveL Target_3090,v100,z1,Marcador\WObj:=Pastel;
        MoveL Target_3100,v100,z1,Marcador\WObj:=Pastel;
        MoveL Target_3110,v100,z1,Marcador\WObj:=Pastel;
        MoveL Target_3120,v100,z1,Marcador\WObj:=Pastel;
        MoveL Target_3130,v100,z1,Marcador\WObj:=Pastel;
        MoveL Target_3140,v100,z1,Marcador\WObj:=Pastel;
        MoveL Target_3150,v100,z1,Marcador\WObj:=Pastel;
        MoveL Target_3160,v100,z1,Marcador\WObj:=Pastel;
        MoveL Target_3170,v100,z1,Marcador\WObj:=Pastel;
        MoveL Target_3180,v100,z1,Marcador\WObj:=Pastel;
        MoveL Target_3190,v100,z1,Marcador\WObj:=Pastel;
        MoveL Target_3200,v100,z1,Marcador\WObj:=Pastel;
        MoveL Target_3210,v100,z1,Marcador\WObj:=Pastel;
        MoveL Target_3220,v100,z1,Marcador\WObj:=Pastel;
        MoveL Target_3230,v100,z1,Marcador\WObj:=Pastel;
        MoveL Target_3240,v100,z1,Marcador\WObj:=Pastel;
        MoveL Target_3250,v100,z1,Marcador\WObj:=Pastel;
        MoveL Target_3260,v100,z1,Marcador\WObj:=Pastel;
        MoveL Target_3270,v100,z1,Marcador\WObj:=Pastel;
        MoveL Target_3280,v100,z1,Marcador\WObj:=Pastel;
        MoveL Target_3290,v100,z1,Marcador\WObj:=Pastel;
        MoveL Target_3300,v100,z1,Marcador\WObj:=Pastel;
        MoveL Target_3310,v100,z1,Marcador\WObj:=Pastel;
        MoveL Target_3320,v100,z1,Marcador\WObj:=Pastel;
        MoveL Target_3330,v100,z1,Marcador\WObj:=Pastel;
        MoveL Target_3340,v100,z1,Marcador\WObj:=Pastel;
        MoveL Target_3350,v100,z1,Marcador\WObj:=Pastel;
        MoveL Target_3360,v100,z1,Marcador\WObj:=Pastel;
        MoveL Target_3370,v100,z1,Marcador\WObj:=Pastel;
        MoveL Target_3380,v100,z1,Marcador\WObj:=Pastel;
        MoveL Target_3390,v100,z1,Marcador\WObj:=Pastel;
        MoveL Target_3400,v100,z1,Marcador\WObj:=Pastel;
        MoveL Target_3410,v100,z1,Marcador\WObj:=Pastel;
        MoveL Target_3420,v100,z1,Marcador\WObj:=Pastel;
        MoveL Target_3430,v100,z1,Marcador\WObj:=Pastel;
        MoveL Target_3440,v100,z1,Marcador\WObj:=Pastel;
        MoveL Target_3450,v100,z1,Marcador\WObj:=Pastel;
        MoveL Target_3460,v100,z1,Marcador\WObj:=Pastel;
        MoveL Target_3470,v100,z1,Marcador\WObj:=Pastel;
        MoveL Target_3480,v100,z1,Marcador\WObj:=Pastel;
        MoveL Target_3490,v100,z1,Marcador\WObj:=Pastel;
        MoveL Target_3500,v100,z1,Marcador\WObj:=Pastel;
        MoveL Target_3510,v100,z1,Marcador\WObj:=Pastel;
        MoveL Target_3520,v100,z1,Marcador\WObj:=Pastel;
        MoveL Target_3530,v100,z1,Marcador\WObj:=Pastel;
        MoveL Target_3540,v100,z1,Marcador\WObj:=Pastel;
        MoveL Target_3550,v100,z1,Marcador\WObj:=Pastel;
        MoveL Target_3560,v100,z1,Marcador\WObj:=Pastel;
        MoveL Target_3570,v100,z1,Marcador\WObj:=Pastel;
        MoveL Target_3580,v100,z1,Marcador\WObj:=Pastel;
        MoveL Target_3590,v100,z1,Marcador\WObj:=Pastel;
        MoveL Target_3600,v100,z1,Marcador\WObj:=Pastel;
        MoveL Target_3610,v100,z1,Marcador\WObj:=Pastel;
    ENDPROC
    PROC DKYMA()
        MoveL Target_3620,v100,z1,Marcador\WObj:=Pastel;
        MoveL Target_3630,v100,z1,Marcador\WObj:=Pastel;
        MoveL Target_3640,v100,z1,Marcador\WObj:=Pastel;
        MoveL Target_3650,v100,z1,Marcador\WObj:=Pastel;
        MoveL Target_3660,v100,z1,Marcador\WObj:=Pastel;
        MoveL Target_3670,v100,z1,Marcador\WObj:=Pastel;
        MoveL Target_3680,v100,z1,Marcador\WObj:=Pastel;
        MoveL Target_3690,v100,z1,Marcador\WObj:=Pastel;
        MoveL Target_3930,v100,z1,Marcador\WObj:=Pastel;
        MoveL Target_3700,v100,z1,Marcador\WObj:=Pastel;
        MoveL Target_3710,v100,z1,Marcador\WObj:=Pastel;
        MoveL Target_3720,v100,z1,Marcador\WObj:=Pastel;
        MoveL Target_3730,v100,z1,Marcador\WObj:=Pastel;
        MoveL Target_3740,v100,z1,Marcador\WObj:=Pastel;
        MoveL Target_3750,v100,z1,Marcador\WObj:=Pastel;
        MoveL Target_3760,v100,z1,Marcador\WObj:=Pastel;
        MoveL Target_3770,v100,z1,Marcador\WObj:=Pastel;
        MoveL Target_3780,v100,z1,Marcador\WObj:=Pastel;
        MoveL Target_3790,v100,z1,Marcador\WObj:=Pastel;
        MoveL Target_3800,v100,z1,Marcador\WObj:=Pastel;
        MoveL Target_3810,v100,z1,Marcador\WObj:=Pastel;
        MoveL Target_3820,v100,z1,Marcador\WObj:=Pastel;
        MoveL Target_3830,v100,z1,Marcador\WObj:=Pastel;
        MoveL Target_3840,v100,z1,Marcador\WObj:=Pastel;
        MoveL Target_3850,v100,z1,Marcador\WObj:=Pastel;
        MoveL Target_3860,v100,z1,Marcador\WObj:=Pastel;
        MoveL Target_3870,v100,z1,Marcador\WObj:=Pastel;
        MoveL Target_3880,v100,z1,Marcador\WObj:=Pastel;
        MoveL Target_3890,v100,z1,Marcador\WObj:=Pastel;
        MoveL Target_3900,v100,z1,Marcador\WObj:=Pastel;
        MoveL Target_3910,v100,z1,Marcador\WObj:=Pastel;
        MoveL Target_3920,v100,z1,Marcador\WObj:=Pastel;
        MoveL Target_3930,v100,z1,Marcador\WObj:=Pastel;
        MoveL Target_3940,v100,z1,Marcador\WObj:=Pastel;
    ENDPROC

    PROC Homming()
        CONST num tol := 0.5;
        VAR jointtarget jt;
        jt := CJointT();
        IF  Abs(jt.robax.rax_1) < tol AND
            Abs(jt.robax.rax_2) < tol AND
            Abs(jt.robax.rax_3) < tol AND
            Abs(jt.robax.rax_4) < tol AND
            Abs(jt.robax.rax_5) < tol AND
            Abs(jt.robax.rax_6) < tol THEN

            TPWrite "Robot en home articular (Aprox 0)";
        ELSE
            TPWrite "Robot no está en home";
            TPWrite "Yendo a Home";
            MoveL HOME,v100,z1,Marcador\WObj:=Pastel;
            MoveAbsJ home0, v500, fine, Marcador;
            TPWrite "Robot en Home";
        ENDIF


